   DATA[75,2] := 2.0;
   DATA[75,3] := 2.0;
   DATA[75,4] := 262.0161;
   DATA[75,5] := 8.391951;
   DATA[75,6] := 328.4286;
   DATA[75,7] := 2.440137;
   DATA[75,8] := 2.0;
   DATA[75,9] := 2.0;
   DATA[75,10] := 2.0;
   DATA[75,11] := 19.59472;
   DATA[75,12] := 2.21055;
   DATA[75,13] := 960.3307;
   DATA[75,14] := 1.0;
   DATA[75,15] := 2.0;
   DATA[75,16] := 1.0;
   DATA[75,17] := 1.0;
   DATA[75,18] := 1.0;
   DATA[75,19] := 2.0;
   DATA[75,20] := 148.808;
   DATA[75,21] := 156.242;
   DATA[75,22] := 1.720309;
   DATA[75,23] := 947.757;
   DATA[75,24] := 2.0;
   DATA[75,25] := 2.0;
   DATA[75,26] := 7.878621;
   DATA[75,27] := 145.0397;
   DATA[75,28] := 264.4194;
   DATA[75,29] := 12.03538;
   DATA[75,30] := 1.729428;
   DATA[75,31] := 1.291533;
   DATA[75,32] := 0.736421;
   DATA[75,33] := 0.3065689;
   DATA[75,34] := 2.0;
   DATA[75,35] := 251.2657;
   DATA[75,36] := 1.665972;
   DATA[75,37] := 189.9833;
   DATA[75,38] := 0.000128152;
   DATA[75,39] := 1.0;
   DATA[76,0] := 2.44179;
   DATA[76,1] := 524.6916;
   DATA[76,2] := 2.0;
   DATA[76,3] := 2.0;
   DATA[76,4] := 262.0161;
   DATA[76,5] := 8.391951;
   DATA[76,6] := 328.4286;
   DATA[76,7] := 2.440137;
   DATA[76,8] := 2.0;
   DATA[76,9] := 2.0;
   DATA[76,10] := 2.0;
   DATA[76,11] := 19.62354;
   DATA[76,12] := 2.21055;
   DATA[76,13] := 959.9702;
   DATA[76,14] := 1.0;
   DATA[76,15] := 2.0;
   DATA[76,16] := 1.0;
   DATA[76,17] := 1.0;
   DATA[76,18] := 1.0;
   DATA[76,19] := 2.0;
   DATA[76,20] := 148.808;
   DATA[76,21] := 156.242;
   DATA[76,22] := 1.719796;
   DATA[76,23] := 948.2184;
   DATA[76,24] := 2.0;
   DATA[76,25] := 2.0;
   DATA[76,26] := 7.878621;
   DATA[76,27] := 145.0397;
   DATA[76,28] := 264.4194;
   DATA[76,29] := 12.03538;
   DATA[76,30] := 1.726096;
   DATA[76,31] := 1.303446;
   DATA[76,32] := 0.736421;
   DATA[76,33] := 0.3065689;
   DATA[76,34] := 2.0;
   DATA[76,35] := 251.2657;
   DATA[76,36] := 1.665972;
   DATA[76,37] := 189.9833;
   DATA[76,38] := 0.000128152;
   DATA[76,39] := 1.0;
   DATA[77,0] := 2.431221;
   DATA[77,1] := 525.0842;
   DATA[77,2] := 2.0;
   DATA[77,3] := 2.0;
   DATA[77,4] := 262.0161;
   DATA[77,5] := 8.391951;
   DATA[77,6] := 328.4286;
   DATA[77,7] := 2.440137;
   DATA[77,8] := 2.0;
   DATA[77,9] := 2.0;
   DATA[77,10] := 2.0;
   DATA[77,11] := 19.64274;
   DATA[77,12] := 2.21055;
   DATA[77,13] := 960.0103;
   DATA[77,14] := 1.0;
   DATA[77,15] := 2.0;
   DATA[77,16] := 1.0;
   DATA[77,17] := 1.0;
   DATA[77,18] := 1.0;
   DATA[77,19] := 2.0;
   DATA[77,20] := 148.808;
   DATA[77,21] := 156.242;
   DATA[77,22] := 1.718515;
   DATA[77,23] := 948.6029;
   DATA[77,24] := 2.0;
   DATA[77,25] := 2.0;
   DATA[77,26] := 7.878621;
   DATA[77,27] := 145.0397;
   DATA[77,28] := 264.4194;
   DATA[77,29] := 12.03538;
   DATA[77,30] := 1.726096;
   DATA[77,31] := 1.311387;
   DATA[77,32] := 0.736421;
   DATA[77,33] := 0.3068891;
   DATA[77,34] := 2.0;
   DATA[77,35] := 250.9933;
   DATA[77,36] := 1.665972;
   DATA[77,37] := 189.8071;
   DATA[77,38] := 0.000128152;
   DATA[77,39] := 1.0;
   DATA[78,0] := 2.421932;
   DATA[78,1] := 525.2411;
   DATA[78,2] := 2.0;
   DATA[78,3] := 2.0;
   DATA[78,4] := 262.0161;
   DATA[78,5] := 8.391951;
   DATA[78,6] := 328.4286;
   DATA[78,7] := 2.440137;
   DATA[78,8] := 2.0;
   DATA[78,9] := 2.0;
   DATA[78,10] := 2.0;
   DATA[78,11] := 19.64274;
   DATA[78,12] := 2.208756;
   DATA[78,13] := 960.1304;
   DATA[78,14] := 1.0;
   DATA[78,15] := 2.0;
   DATA[78,16] := 1.0;
   DATA[78,17] := 1.0;
   DATA[78,18] := 1.0;
   DATA[78,19] := 2.0;
   DATA[78,20] := 148.808;
   DATA[78,21] := 156.242;
   DATA[78,22] := 1.718515;
   DATA[78,23] := 948.5645;
   DATA[78,24] := 2.0;
   DATA[78,25] := 2.0;
   DATA[78,26] := 7.878621;
   DATA[78,27] := 145.0397;
   DATA[78,28] := 264.2912;
   DATA[78,29] := 12.03538;
   DATA[78,30] := 1.725968;
   DATA[78,31] := 1.306008;
   DATA[78,32] := 0.736421;
   DATA[78,33] := 0.3068891;
   DATA[78,34] := 2.0;
   DATA[78,35] := 250.9933;
   DATA[78,36] := 1.665972;
   DATA[78,37] := 189.6629;
   DATA[78,38] := 0.000128152;
   DATA[78,39] := 1.0;
   DATA[79,0] := 2.420011;
   DATA[79,1] := 525.5159;
   DATA[79,2] := 2.0;
   DATA[79,3] := 2.0;
   DATA[79,4] := 262.0161;
   DATA[79,5] := 8.391951;
   DATA[79,6] := 328.4286;
   DATA[79,7] := 2.440137;
   DATA[79,8] := 2.0;
   DATA[79,9] := 2.0;
   DATA[79,10] := 2.0;
   DATA[79,11] := 19.64274;
   DATA[79,12] := 2.208756;
   DATA[79,13] := 959.9702;
   DATA[79,14] := 1.0;
   DATA[79,15] := 2.0;
   DATA[79,16] := 1.0;
   DATA[79,17] := 1.0;
   DATA[79,18] := 1.0;
   DATA[79,19] := 2.0;
   DATA[79,20] := 148.808;
   DATA[79,21] := 156.242;
   DATA[79,22] := 1.720309;
   DATA[79,23] := 948.7952;
   DATA[79,24] := 2.0;
   DATA[79,25] := 2.0;
   DATA[79,26] := 7.878621;
   DATA[79,27] := 145.1679;
   DATA[79,28] := 264.2912;
   DATA[79,29] := 12.03538;
   DATA[79,30] := 1.724814;
   DATA[79,31] := 1.306904;
   DATA[79,32] := 0.7353967;
   DATA[79,33] := 0.3068891;
   DATA[79,34] := 2.0;
   DATA[79,35] := 250.9933;
   DATA[79,36] := 1.665972;
   DATA[79,37] := 189.6629;
   DATA[79,38] := 0.000128152;
   DATA[79,39] := 1.0;
   DATA[80,0] := 2.447875;
   DATA[80,1] := 525.3196;
   DATA[80,2] := 2.0;
   DATA[80,3] := 2.0;
   DATA[80,4] := 262.0161;
   DATA[80,5] := 8.394835;
   DATA[80,6] := 328.4286;
   DATA[80,7] := 2.440137;
   DATA[80,8] := 2.0;
   DATA[80,9] := 2.0;
   DATA[80,10] := 2.0;
   DATA[80,11] := 19.65555;
   DATA[80,12] := 2.208756;
   DATA[80,13] := 960.3708;
   DATA[80,14] := 1.0;
   DATA[80,15] := 2.0;
   DATA[80,16] := 1.0;
   DATA[80,17] := 1.0;
   DATA[80,18] := 1.0;
   DATA[80,19] := 2.0;
   DATA[80,20] := 148.808;
   DATA[80,21] := 156.242;
   DATA[80,22] := 1.720309;
   DATA[80,23] := 948.9105;
   DATA[80,24] := 2.0;
   DATA[80,25] := 2.0;
   DATA[80,26] := 7.878621;
   DATA[80,27] := 145.2448;
   DATA[80,28] := 264.2912;
   DATA[80,29] := 12.03538;
   DATA[80,30] := 1.724814;
   DATA[80,31] := 1.297938;
   DATA[80,32] := 0.7353967;
   DATA[80,33] := 0.3068891;
   DATA[80,34] := 2.0;
   DATA[80,35] := 250.9933;
   DATA[80,36] := 1.665972;
   DATA[80,37] := 189.6629;
   DATA[80,38] := 0.000128152;
   DATA[80,39] := 1.0;
   DATA[81,0] := 2.500721;
   DATA[81,1] := 526.0262;
   DATA[81,2] := 2.0;
   DATA[81,3] := 2.0;
   DATA[81,4] := 262.0161;
   DATA[81,5] := 8.394835;
   DATA[81,6] := 328.4286;
   DATA[81,7] := 2.440137;
   DATA[81,8] := 2.0;
   DATA[81,9] := 2.0;
   DATA[81,10] := 2.0;
   DATA[81,11] := 19.65555;
   DATA[81,12] := 2.208756;
   DATA[81,13] := 960.2506;
   DATA[81,14] := 1.0;
   DATA[81,15] := 2.0;
   DATA[81,16] := 1.0;
   DATA[81,17] := 1.0;
   DATA[81,18] := 1.0;
   DATA[81,19] := 2.0;
   DATA[81,20] := 148.808;
   DATA[81,21] := 156.242;
   DATA[81,22] := 1.720309;
   DATA[81,23] := 949.1028;
   DATA[81,24] := 2.0;
   DATA[81,25] := 2.0;
   DATA[81,26] := 7.878621;
   DATA[81,27] := 145.2448;
   DATA[81,28] := 264.2592;
   DATA[81,29] := 12.03538;
   DATA[81,30] := 1.724814;
   DATA[81,31] := 1.292174;
   DATA[81,32] := 0.7353967;
   DATA[81,33] := 0.3066329;
   DATA[81,34] := 2.0;
   DATA[81,35] := 250.9933;
   DATA[81,36] := 1.569859;
   DATA[81,37] := 189.6629;
   DATA[81,38] := 0.000128152;
   DATA[81,39] := 1.0;
   DATA[82,0] := 2.543958;
   DATA[82,1] := 526.4973;
   DATA[82,2] := 2.0;
   DATA[82,3] := 2.0;
   DATA[82,4] := 262.0161;
   DATA[82,5] := 8.394835;
   DATA[82,6] := 328.4286;
   DATA[82,7] := 2.440137;
   DATA[82,8] := 2.0;
   DATA[82,9] := 2.0;
   DATA[82,10] := 2.0;
   DATA[82,11] := 19.65555;
   DATA[82,12] := 2.208756;
   DATA[82,13] := 960.0904;
   DATA[82,14] := 1.0;
   DATA[82,15] := 2.0;
   DATA[82,16] := 1.0;
   DATA[82,17] := 1.0;
   DATA[82,18] := 1.0;
   DATA[82,19] := 2.0;
   DATA[82,20] := 148.808;
   DATA[82,21] := 156.242;
   DATA[82,22] := 1.718643;
   DATA[82,23] := 949.1797;
   DATA[82,24] := 2.0;
   DATA[82,25] := 2.0;
   DATA[82,26] := 7.878621;
   DATA[82,27] := 145.2448;
   DATA[82,28] := 264.2592;
   DATA[82,29] := 12.03538;
   DATA[82,30] := 1.724814;
   DATA[82,31] := 1.288971;
   DATA[82,32] := 0.7353967;
   DATA[82,33] := 0.3065048;
   DATA[82,34] := 2.0;
   DATA[82,35] := 250.9933;
   DATA[82,36] := 1.569859;
   DATA[82,37] := 189.6629;
   DATA[82,38] := 0.000128152;
   DATA[82,39] := 1.0;
   DATA[83,0] := 2.570861;
   DATA[83,1] := 526.8898;
   DATA[83,2] := 2.0;
   DATA[83,3] := 2.0;
   DATA[83,4] := 262.0161;
   DATA[83,5] := 8.394835;
   DATA[83,6] := 328.4286;
   DATA[83,7] := 2.441034;
   DATA[83,8] := 2.0;
   DATA[83,9] := 2.0;
   DATA[83,10] := 2.0;
   DATA[83,11] := 19.65555;
   DATA[83,12] := 2.208756;
   DATA[83,13] := 959.8901;
   DATA[83,14] := 1.0;
   DATA[83,15] := 2.0;
   DATA[83,16] := 1.0;
   DATA[83,17] := 1.0;
   DATA[83,18] := 1.0;
   DATA[83,19] := 2.0;
   DATA[83,20] := 148.808;
   DATA[83,21] := 156.242;
   DATA[83,22] := 1.718643;
   DATA[83,23] := 949.2181;
   DATA[83,24] := 2.0;
   DATA[83,25] := 2.0;
   DATA[83,26] := 7.878621;
   DATA[83,27] := 145.2448;
   DATA[83,28] := 264.2592;
   DATA[83,29] := 12.03538;
   DATA[83,30] := 1.724814;
   DATA[83,31] := 1.282311;
   DATA[83,32] := 0.7353967;
   DATA[83,33] := 0.3065048;
   DATA[83,34] := 2.0;
   DATA[83,35] := 250.9933;
   DATA[83,36] := 1.569859;
   DATA[83,37] := 189.6629;
   DATA[83,38] := 0.000128152;
   DATA[83,39] := 1.0;
   DATA[84,0] := 2.614739;
   DATA[84,1] := 527.2038;
   DATA[84,2] := 2.0;
   DATA[84,3] := 2.0;
   DATA[84,4] := 262.0161;
   DATA[84,5] := 8.394835;
   DATA[84,6] := 328.4286;
   DATA[84,7] := 2.441034;
   DATA[84,8] := 2.0;
   DATA[84,9] := 2.0;
   DATA[84,10] := 2.0;
   DATA[84,11] := 19.65555;
   DATA[84,12] := 2.208756;
   DATA[84,13] := 959.8901;
   DATA[84,14] := 1.0;
   DATA[84,15] := 2.0;
   DATA[84,16] := 1.0;
   DATA[84,17] := 1.0;
   DATA[84,18] := 1.0;
   DATA[84,19] := 2.0;
   DATA[84,20] := 148.808;
   DATA[84,21] := 156.242;
   DATA[84,22] := 1.718643;
   DATA[84,23] := 949.8718;
   DATA[84,24] := 2.0;
   DATA[84,25] := 2.0;
   DATA[84,26] := 7.878621;
   DATA[84,27] := 145.1423;
   DATA[84,28] := 264.2592;
   DATA[84,29] := 12.03538;
   DATA[84,30] := 1.724814;
   DATA[84,31] := 1.27898;
   DATA[84,32] := 0.7353967;
   DATA[84,33] := 0.3065048;
   DATA[84,34] := 2.0;
   DATA[84,35] := 250.9933;
   DATA[84,36] := 1.569859;
   DATA[84,37] := 189.6629;
   DATA[84,38] := 0.000128152;
   DATA[84,39] := 1.0;
   DATA[85,0] := 2.645806;
   DATA[85,1] := 527.3608;
   DATA[85,2] := 2.0;
   DATA[85,3] := 2.0;
   DATA[85,4] := 262.2084;
   DATA[85,5] := 8.394835;
   DATA[85,6] := 328.4286;
   DATA[85,7] := 2.441034;
   DATA[85,8] := 2.0;
   DATA[85,9] := 2.0;
   DATA[85,10] := 2.0;
   DATA[85,11] := 19.65555;
   DATA[85,12] := 2.208756;
   DATA[85,13] := 960.0103;
   DATA[85,14] := 1.0;
   DATA[85,15] := 2.0;
   DATA[85,16] := 1.0;
   DATA[85,17] := 1.0;
   DATA[85,18] := 1.0;
   DATA[85,19] := 2.0;
   DATA[85,20] := 148.808;
   DATA[85,21] := 156.0882;
   DATA[85,22] := 1.720693;
   DATA[85,23] := 950.0641;
   DATA[85,24] := 2.0;
   DATA[85,25] := 2.0;
   DATA[85,26] := 7.878621;
   DATA[85,27] := 144.9885;
   DATA[85,28] := 264.2592;
   DATA[85,29] := 12.03538;
   DATA[85,30] := 1.724814;
   DATA[85,31] := 1.27232;
   DATA[85,32] := 0.7353967;
   DATA[85,33] := 0.3065048;
   DATA[85,34] := 2.0;
   DATA[85,35] := 250.9933;
   DATA[85,36] := 1.569859;
   DATA[85,37] := 189.7751;
   DATA[85,38] := 0.000128152;
   DATA[85,39] := 1.0;
   DATA[86,0] := 2.665023;
   DATA[86,1] := 527.4786;
   DATA[86,2] := 2.0;
   DATA[86,3] := 2.0;
   DATA[86,4] := 262.2084;
   DATA[86,5] := 8.394835;
   DATA[86,6] := 328.4286;
   DATA[86,7] := 2.441034;
   DATA[86,8] := 2.0;
   DATA[86,9] := 2.0;
   DATA[86,10] := 2.0;
   DATA[86,11] := 19.65555;
   DATA[86,12] := 2.208756;
   DATA[86,13] := 959.8901;
   DATA[86,14] := 1.0;
   DATA[86,15] := 2.0;
   DATA[86,16] := 1.0;
   DATA[86,17] := 1.0;
   DATA[86,18] := 1.0;
   DATA[86,19] := 2.0;
   DATA[86,20] := 148.808;
   DATA[86,21] := 156.0882;
   DATA[86,22] := 1.720693;
   DATA[86,23] := 950.1794;
   DATA[86,24] := 2.0;
   DATA[86,25] := 2.0;
   DATA[86,26] := 7.878621;
   DATA[86,27] := 144.9885;
   DATA[86,28] := 264.2592;
   DATA[86,29] := 12.03538;
   DATA[86,30] := 1.724814;
   DATA[86,31] := 1.270398;
   DATA[86,32] := 0.7353967;
   DATA[86,33] := 0.3065048;
   DATA[86,34] := 2.0;
   DATA[86,35] := 250.9933;
   DATA[86,36] := 1.569859;
   DATA[86,37] := 189.7751;
   DATA[86,38] := 0.000128152;
   DATA[86,39] := 1.0;
   DATA[87,0] := 2.666944;
   DATA[87,1] := 527.7534;
   DATA[87,2] := 2.0;
   DATA[87,3] := 2.0;
   DATA[87,4] := 262.2084;
   DATA[87,5] := 8.393553;
   DATA[87,6] := 328.4286;
   DATA[87,7] := 2.441547;
   DATA[87,8] := 2.0;
   DATA[87,9] := 2.0;
   DATA[87,10] := 2.0;
   DATA[87,11] := 19.65555;
   DATA[87,12] := 2.208756;
   DATA[87,13] := 959.5296;
   DATA[87,14] := 1.0;
   DATA[87,15] := 2.0;
   DATA[87,16] := 1.0;
   DATA[87,17] := 1.0;
   DATA[87,18] := 1.0;
   DATA[87,19] := 2.0;
   DATA[87,20] := 148.808;
   DATA[87,21] := 156.0882;
   DATA[87,22] := 1.720693;
   DATA[87,23] := 950.0641;
   DATA[87,24] := 2.0;
   DATA[87,25] := 2.0;
   DATA[87,26] := 7.878621;
   DATA[87,27] := 144.9885;
   DATA[87,28] := 264.2592;
   DATA[87,29] := 12.30454;
   DATA[87,30] := 1.724814;
   DATA[87,31] := 1.270398;
   DATA[87,32] := 0.7353967;
   DATA[87,33] := 0.3065048;
   DATA[87,34] := 2.0;
   DATA[87,35] := 250.9933;
   DATA[87,36] := 1.569859;
   DATA[87,37] := 189.7751;
   DATA[87,38] := 0.000128152;
   DATA[87,39] := 1.0;
   DATA[88,0] := 2.6394;
   DATA[88,1] := 528.2244;
   DATA[88,2] := 2.0;
   DATA[88,3] := 2.0;
   DATA[88,4] := 262.2084;
   DATA[88,5] := 8.391951;
   DATA[88,6] := 328.4286;
   DATA[88,7] := 2.443597;
   DATA[88,8] := 2.0;
   DATA[88,9] := 2.0;
   DATA[88,10] := 2.0;
   DATA[88,11] := 19.65555;
   DATA[88,12] := 2.209653;
   DATA[88,13] := 959.4896;
   DATA[88,14] := 1.0;
   DATA[88,15] := 2.0;
   DATA[88,16] := 1.0;
   DATA[88,17] := 1.0;
   DATA[88,18] := 1.0;
   DATA[88,19] := 2.0;
   DATA[88,20] := 148.808;
   DATA[88,21] := 156.0882;
   DATA[88,22] := 1.720693;
   DATA[88,23] := 950.2563;
   DATA[88,24] := 2.0;
   DATA[88,25] := 2.0;
   DATA[88,26] := 7.878621;
   DATA[88,27] := 144.9885;
   DATA[88,28] := 264.2592;
   DATA[88,29] := 12.30454;
   DATA[88,30] := 1.727378;
   DATA[88,31] := 1.284232;
   DATA[88,32] := 0.7353967;
   DATA[88,33] := 0.3065048;
   DATA[88,34] := 2.0;
   DATA[88,35] := 250.9933;
   DATA[88,36] := 1.569859;
   DATA[88,37] := 189.7751;
   DATA[88,38] := 0.000128152;
   DATA[88,39] := 1.0;
   DATA[89,0] := 2.620824;
   DATA[89,1] := 527.8711;
   DATA[89,2] := 2.0;
   DATA[89,3] := 2.0;
   DATA[89,4] := 261.9841;
   DATA[89,5] := 8.391951;
   DATA[89,6] := 328.4286;
   DATA[89,7] := 2.444751;
   DATA[89,8] := 2.0;
   DATA[89,9] := 2.0;
   DATA[89,10] := 2.0;
   DATA[89,11] := 19.60433;
   DATA[89,12] := 2.209653;
   DATA[89,13] := 959.5697;
   DATA[89,14] := 1.0;
   DATA[89,15] := 2.0;
   DATA[89,16] := 1.0;
   DATA[89,17] := 1.0;
   DATA[89,18] := 1.0;
   DATA[89,19] := 2.0;
   DATA[89,20] := 148.808;
   DATA[89,21] := 156.0882;
   DATA[89,22] := 1.719924;
   DATA[89,23] := 950.5255;
   DATA[89,24] := 2.0;
   DATA[89,25] := 2.0;
   DATA[89,26] := 7.878621;
   DATA[89,27] := 144.9885;
   DATA[89,28] := 264.2592;
   DATA[89,29] := 12.30454;
   DATA[89,30] := 1.727378;
   DATA[89,31] := 1.290765;
   DATA[89,32] := 0.7353967;
   DATA[89,33] := 0.3065048;
   DATA[89,34] := 2.0;
   DATA[89,35] := 250.9933;
   DATA[89,36] := 1.569859;
   DATA[89,37] := 189.7751;
   DATA[89,38] := 0.000128152;
   DATA[89,39] := 1.0;
   DATA[90,0] := 2.61634;
   DATA[90,1] := 528.0281;
   DATA[90,2] := 2.0;
   DATA[90,3] := 2.0;
   DATA[90,4] := 261.9841;
   DATA[90,5] := 8.391951;
   DATA[90,6] := 328.4286;
   DATA[90,7] := 2.444751;
   DATA[90,8] := 2.0;
   DATA[90,9] := 2.0;
   DATA[90,10] := 2.0;
   DATA[90,11] := 19.60433;
   DATA[90,12] := 2.209653;
   DATA[90,13] := 959.5697;
   DATA[90,14] := 1.0;
   DATA[90,15] := 2.0;
   DATA[90,16] := 1.0;
   DATA[90,17] := 1.0;
   DATA[90,18] := 1.0;
   DATA[90,19] := 2.0;
   DATA[90,20] := 148.808;
   DATA[90,21] := 156.0882;
   DATA[90,22] := 1.719284;
   DATA[90,23] := 950.6409;
   DATA[90,24] := 2.0;
   DATA[90,25] := 2.0;
   DATA[90,26] := 7.878621;
   DATA[90,27] := 145.1166;
   DATA[90,28] := 264.2592;
   DATA[90,29] := 12.30454;
   DATA[90,30] := 1.727378;
   DATA[90,31] := 1.285385;
   DATA[90,32] := 0.7353967;
   DATA[90,33] := 0.3065048;
   DATA[90,34] := 2.0;
   DATA[90,35] := 250.9933;
   DATA[90,36] := 1.681991;
   DATA[90,37] := 189.7751;
   DATA[90,38] := 0.000128152;
   DATA[90,39] := 1.0;
   DATA[91,0] := 2.61602;
   DATA[91,1] := 527.7534;
   DATA[91,2] := 2.0;
   DATA[91,3] := 2.0;
   DATA[91,4] := 261.9841;
   DATA[91,5] := 8.391951;
   DATA[91,6] := 328.4286;
   DATA[91,7] := 2.444751;
   DATA[91,8] := 2.0;
   DATA[91,9] := 2.0;
   DATA[91,10] := 2.0;
   DATA[91,11] := 19.60433;
   DATA[91,12] := 2.212215;
   DATA[91,13] := 959.4095;
   DATA[91,14] := 1.0;
   DATA[91,15] := 2.0;
   DATA[91,16] := 1.0;
   DATA[91,17] := 1.0;
   DATA[91,18] := 1.0;
   DATA[91,19] := 2.0;
   DATA[91,20] := 148.808;
   DATA[91,21] := 156.0882;
   DATA[91,22] := 1.719284;
   DATA[91,23] := 950.8331;
   DATA[91,24] := 2.0;
   DATA[91,25] := 2.0;
   DATA[91,26] := 7.878621;
   DATA[91,27] := 145.1679;
   DATA[91,28] := 264.2592;
   DATA[91,29] := 12.30454;
   DATA[91,30] := 1.727378;
   DATA[91,31] := 1.288843;
   DATA[91,32] := 0.7353967;
   DATA[91,33] := 0.3065048;
   DATA[91,34] := 2.0;
   DATA[91,35] := 250.9933;
   DATA[91,36] := 1.681991;
   DATA[91,37] := 189.7751;
   DATA[91,38] := 0.000128152;
   DATA[91,39] := 1.0;
   DATA[92,0] := 2.609294;
   DATA[92,1] := 527.4393;
   DATA[92,2] := 2.0;
   DATA[92,3] := 2.0;
   DATA[92,4] := 261.9841;
   DATA[92,5] := 8.391951;
   DATA[92,6] := 328.4286;
   DATA[92,7] := 2.443085;
   DATA[92,8] := 2.0;
   DATA[92,9] := 2.0;
   DATA[92,10] := 2.0;
   DATA[92,11] := 19.64274;
   DATA[92,12] := 2.212215;
   DATA[92,13] := 959.77;
   DATA[92,14] := 1.0;
   DATA[92,15] := 2.0;
   DATA[92,16] := 1.0;
   DATA[92,17] := 1.0;
   DATA[92,18] := 1.0;
   DATA[92,19] := 2.0;
   DATA[92,20] := 148.808;
   DATA[92,21] := 156.0882;
   DATA[92,22] := 1.718387;
   DATA[92,23] := 950.8716;
   DATA[92,24] := 2.0;
   DATA[92,25] := 2.0;
   DATA[92,26] := 7.878621;
   DATA[92,27] := 145.1679;
   DATA[92,28] := 264.2592;
   DATA[92,29] := 12.30454;
   DATA[92,30] := 1.727378;
   DATA[92,31] := 1.278468;
   DATA[92,32] := 0.7353967;
   DATA[92,33] := 0.3065048;
   DATA[92,34] := 2.0;
   DATA[92,35] := 250.9933;
   DATA[92,36] := 1.681991;
   DATA[92,37] := 189.7751;
   DATA[92,38] := 0.000128152;
   DATA[92,39] := 1.0;
   DATA[93,0] := 2.584313;
   DATA[93,1] := 527.2823;
   DATA[93,2] := 2.0;
   DATA[93,3] := 2.0;
   DATA[93,4] := 261.9841;
   DATA[93,5] := 8.391951;
   DATA[93,6] := 328.4286;
   DATA[93,7] := 2.442316;
   DATA[93,8] := 2.0;
   DATA[93,9] := 2.0;
   DATA[93,10] := 2.0;
   DATA[93,11] := 19.65875;
   DATA[93,12] := 2.212343;
   DATA[93,13] := 960.0904;
   DATA[93,14] := 1.0;
   DATA[93,15] := 2.0;
   DATA[93,16] := 1.0;
   DATA[93,17] := 1.0;
   DATA[93,18] := 1.0;
   DATA[93,19] := 2.0;
   DATA[93,20] := 148.808;
   DATA[93,21] := 156.0882;
   DATA[93,22] := 1.716849;
   DATA[93,23] := 951.0638;
   DATA[93,24] := 2.0;
   DATA[93,25] := 2.0;
   DATA[93,26] := 7.877019;
   DATA[93,27] := 145.1679;
   DATA[93,28] := 264.2592;
   DATA[93,29] := 12.30454;
   DATA[93,30] := 1.727378;
   DATA[93,31] := 1.263097;
   DATA[93,32] := 0.7353967;
   DATA[93,33] := 0.3065048;
   DATA[93,34] := 2.0;
   DATA[93,35] := 251.1055;
   DATA[93,36] := 1.649953;
   DATA[93,37] := 189.7751;
   DATA[93,38] := 0.000128152;
   DATA[93,39] := 1.0;
   DATA[94,0] := 2.572463;
   DATA[94,1] := 527.2823;
   DATA[94,2] := 2.0;
   DATA[94,3] := 2.0;
   DATA[94,4] := 261.9841;
   DATA[94,5] := 8.391951;
   DATA[94,6] := 328.4286;
   DATA[94,7] := 2.442188;
   DATA[94,8] := 2.0;
   DATA[94,9] := 2.0;
   DATA[94,10] := 2.0;
   DATA[94,11] := 19.65875;
   DATA[94,12] := 2.212343;
   DATA[94,13] := 960.0103;
   DATA[94,14] := 1.0;
   DATA[94,15] := 2.0;
   DATA[94,16] := 1.0;
   DATA[94,17] := 1.0;
   DATA[94,18] := 1.0;
   DATA[94,19] := 2.0;
   DATA[94,20] := 148.808;
   DATA[94,21] := 156.0882;
   DATA[94,22] := 1.714029;
   DATA[94,23] := 950.8331;
   DATA[94,24] := 2.0;
   DATA[94,25] := 2.0;
   DATA[94,26] := 7.877019;
   DATA[94,27] := 145.1423;
   DATA[94,28] := 264.2592;
   DATA[94,29] := 12.30454;
   DATA[94,30] := 1.727378;
   DATA[94,31] := 1.257589;
   DATA[94,32] := 0.7353967;
   DATA[94,33] := 0.3065048;
   DATA[94,34] := 2.0;
   DATA[94,35] := 251.1055;
   DATA[94,36] := 1.649953;
   DATA[94,37] := 189.7751;
   DATA[94,38] := 0.000128152;
   DATA[94,39] := 1.0;
   DATA[95,0] := 2.554847;
   DATA[95,1] := 527.3608;
   DATA[95,2] := 2.0;
   DATA[95,3] := 2.0;
   DATA[95,4] := 261.9841;
   DATA[95,5] := 8.391951;
   DATA[95,6] := 328.4286;
   DATA[95,7] := 2.442188;
   DATA[95,8] := 2.0;
   DATA[95,9] := 2.0;
   DATA[95,10] := 2.0;
   DATA[95,11] := 19.65875;
   DATA[95,12] := 2.212343;
   DATA[95,13] := 959.9302;
   DATA[95,14] := 1.0;
   DATA[95,15] := 2.0;
   DATA[95,16] := 1.0;
   DATA[95,17] := 1.0;
   DATA[95,18] := 1.0;
   DATA[95,19] := 2.0;
   DATA[95,20] := 148.808;
   DATA[95,21] := 156.0882;
   DATA[95,22] := 1.713261;
   DATA[95,23] := 950.91;
   DATA[95,24] := 2.0;
   DATA[95,25] := 2.0;
   DATA[95,26] := 7.877019;
   DATA[95,27] := 145.1423;
   DATA[95,28] := 264.2592;
   DATA[95,29] := 12.30454;
   DATA[95,30] := 1.727378;
   DATA[95,31] := 1.245549;
   DATA[95,32] := 0.7353967;
   DATA[95,33] := 0.3065048;
   DATA[95,34] := 2.0;
   DATA[95,35] := 251.1055;
   DATA[95,36] := 1.649953;
   DATA[95,37] := 189.7751;
   DATA[95,38] := 0.000128152;
   DATA[95,39] := 1.0;
   DATA[96,0] := 2.542036;
   DATA[96,1] := 526.8113;
   DATA[96,2] := 2.0;
   DATA[96,3] := 2.0;
   DATA[96,4] := 261.9841;
   DATA[96,5] := 8.39163;
   DATA[96,6] := 328.4286;
   DATA[96,7] := 2.442188;
   DATA[96,8] := 2.0;
   DATA[96,9] := 2.0;
   DATA[96,10] := 2.0;
   DATA[96,11] := 19.64594;
   DATA[96,12] := 2.212343;
   DATA[96,13] := 960.2506;
   DATA[96,14] := 1.0;
   DATA[96,15] := 2.0;
   DATA[96,16] := 1.0;
   DATA[96,17] := 1.0;
   DATA[96,18] := 1.0;
   DATA[96,19] := 2.0;
   DATA[96,20] := 148.808;
   DATA[96,21] := 156.0882;
   DATA[96,22] := 1.712876;
   DATA[96,23] := 951.2561;
   DATA[96,24] := 2.0;
   DATA[96,25] := 2.0;
   DATA[96,26] := 7.877019;
   DATA[96,27] := 144.9628;
   DATA[96,28] := 264.2592;
   DATA[96,29] := 12.11228;
   DATA[96,30] := 1.726865;
   DATA[96,31] := 1.256693;
   DATA[96,32] := 0.7353967;
   DATA[96,33] := 0.3065048;
   DATA[96,34] := 2.0;
   DATA[96,35] := 251.1055;
   DATA[96,36] := 1.649953;
   DATA[96,37] := 189.7751;
   DATA[96,38] := 0.000128152;
   DATA[96,39] := 1.0;
   DATA[97,0] := 2.520257;
   DATA[97,1] := 526.5757;
   DATA[97,2] := 2.0;
   DATA[97,3] := 2.0;
   DATA[97,4] := 261.9841;
   DATA[97,5] := 8.39163;
   DATA[97,6] := 328.4286;
   DATA[97,7] := 2.442188;
   DATA[97,8] := 2.0;
   DATA[97,9] := 2.0;
   DATA[97,10] := 2.0;
   DATA[97,11] := 19.62354;
   DATA[97,12] := 2.212343;
   DATA[97,13] := 960.531;
   DATA[97,14] := 1.0;
   DATA[97,15] := 2.0;
   DATA[97,16] := 1.0;
   DATA[97,17] := 1.0;
   DATA[97,18] := 1.0;
   DATA[97,19] := 2.0;
   DATA[97,20] := 148.808;
   DATA[97,21] := 156.0882;
   DATA[97,22] := 1.713261;
   DATA[97,23] := 951.2561;
   DATA[97,24] := 2.0;
   DATA[97,25] := 2.0;
   DATA[97,26] := 7.877019;
   DATA[97,27] := 144.8603;
   DATA[97,28] := 264.2592;
   DATA[97,29] := 12.07383;
   DATA[97,30] := 1.726865;
   DATA[97,31] := 1.265787;
   DATA[97,32] := 0.7353967;
   DATA[97,33] := 0.3074656;
   DATA[97,34] := 2.0;
   DATA[97,35] := 250.9773;
   DATA[97,36] := 1.649953;
   DATA[97,37] := 189.6789;
   DATA[97,38] := 0.000128152;
   DATA[97,39] := 1.0;
   DATA[98,0] := 2.508407;
   DATA[98,1] := 525.8692;
   DATA[98,2] := 2.0;
   DATA[98,3] := 2.0;
   DATA[98,4] := 261.9841;
   DATA[98,5] := 8.39163;
   DATA[98,6] := 328.4286;
   DATA[98,7] := 2.443469;
   DATA[98,8] := 2.0;
   DATA[98,9] := 2.0;
   DATA[98,10] := 2.0;
   DATA[98,11] := 19.62354;
   DATA[98,12] := 2.21055;
   DATA[98,13] := 960.3307;
   DATA[98,14] := 1.0;
   DATA[98,15] := 2.0;
   DATA[98,16] := 1.0;
   DATA[98,17] := 1.0;
   DATA[98,18] := 1.0;
   DATA[98,19] := 2.0;
   DATA[98,20] := 148.808;
   DATA[98,21] := 156.0882;
   DATA[98,22] := 1.715311;
   DATA[98,23] := 951.4099;
   DATA[98,24] := 2.0;
   DATA[98,25] := 2.0;
   DATA[98,26] := 7.877019;
   DATA[98,27] := 144.8603;
   DATA[98,28] := 264.2592;
   DATA[98,29] := 12.07383;
   DATA[98,30] := 1.725583;
   DATA[98,31] := 1.277956;
   DATA[98,32] := 0.7353967;
   DATA[98,33] := 0.3081062;
   DATA[98,34] := 2.0;
   DATA[98,35] := 250.8171;
   DATA[98,36] := 1.649953;
   DATA[98,37] := 189.5027;
   DATA[98,38] := 0.000128152;
   DATA[98,39] := 1.0;
   DATA[99,0] := 2.491112;
   DATA[99,1] := 525.3982;
   DATA[99,2] := 2.0;
   DATA[99,3] := 2.0;
   DATA[99,4] := 261.9841;
   DATA[99,5] := 8.39163;
   DATA[99,6] := 328.4286;
   DATA[99,7] := 2.444751;
   DATA[99,8] := 2.0;
   DATA[99,9] := 2.0;
   DATA[99,10] := 2.0;
   DATA[99,11] := 19.66195;
   DATA[99,12] := 2.209525;
   DATA[99,13] := 960.2106;
   DATA[99,14] := 1.0;
   DATA[99,15] := 2.0;
   DATA[99,16] := 1.0;
   DATA[99,17] := 1.0;
   DATA[99,18] := 1.0;
   DATA[99,19] := 2.0;
   DATA[99,20] := 148.808;
   DATA[99,21] := 156.1907;
   DATA[99,22] := 1.715311;
   DATA[99,23] := 951.2561;
   DATA[99,24] := 2.0;
   DATA[99,25] := 2.0;
   DATA[99,26] := 7.877019;
   DATA[99,27] := 144.8603;
   DATA[99,28] := 264.2592;
   DATA[99,29] := 12.07383;
   DATA[99,30] := 1.725455;
   DATA[99,31] := 1.289484;
   DATA[99,32] := 0.7378293;
   DATA[99,33] := 0.3081062;
   DATA[99,34] := 2.0;
   DATA[99,35] := 250.8171;
   DATA[99,36] := 1.649953;
   DATA[99,37] := 189.5027;
   DATA[99,38] := 0.000128152;
   DATA[99,39] := 1.0;
   DATA[100,0] := 2.476059;
   DATA[100,1] := 525.0842;
   DATA[100,2] := 2.0;
   DATA[100,3] := 2.0;
   DATA[100,4] := 261.9841;
   DATA[100,5] := 8.39163;
   DATA[100,6] := 328.4286;
   DATA[100,7] := 2.444751;
   DATA[100,8] := 2.0;
   DATA[100,9] := 2.0;
   DATA[100,10] := 2.0;
   DATA[100,11] := 19.66195;
   DATA[100,12] := 2.209525;
   DATA[100,13] := 960.3708;
   DATA[100,14] := 1.0;
   DATA[100,15] := 2.0;
   DATA[100,16] := 1.0;
   DATA[100,17] := 1.0;
   DATA[100,18] := 1.0;
   DATA[100,19] := 2.0;
   DATA[100,20] := 148.808;
   DATA[100,21] := 156.1907;
   DATA[100,22] := 1.715311;
   DATA[100,23] := 951.6791;
   DATA[100,24] := 2.0;
   DATA[100,25] := 2.0;
   DATA[100,26] := 7.877019;
   DATA[100,27] := 145.0397;
   DATA[100,28] := 264.2592;
   DATA[100,29] := 12.07383;
   DATA[100,30] := 1.723404;
   DATA[100,31] := 1.286666;
   DATA[100,32] := 0.7378293;
   DATA[100,33] := 0.3084265;
   DATA[100,34] := 2.0;
   DATA[100,35] := 250.8011;
   DATA[100,36] := 1.649953;
   DATA[100,37] := 189.5027;
   DATA[100,38] := 0.000128152;
   DATA[100,39] := 1.0;
   DATA[101,0] := 2.460045;
   DATA[101,1] := 524.8879;
   DATA[101,2] := 2.0;
   DATA[101,3] := 2.0;
   DATA[101,4] := 261.9841;
   DATA[101,5] := 8.39163;
   DATA[101,6] := 328.4286;
   DATA[101,7] := 2.444751;
   DATA[101,8] := 2.0;
   DATA[101,9] := 2.0;
   DATA[101,10] := 2.0;
   DATA[101,11] := 19.55631;
   DATA[101,12] := 2.209525;
   DATA[101,13] := 960.2106;
   DATA[101,14] := 1.0;
   DATA[101,15] := 2.0;
   DATA[101,16] := 1.0;
   DATA[101,17] := 1.0;
   DATA[101,18] := 1.0;
   DATA[101,19] := 2.0;
   DATA[101,20] := 148.808;
   DATA[101,21] := 156.1907;
   DATA[101,22] := 1.717105;
   DATA[101,23] := 951.9867;
   DATA[101,24] := 2.0;
   DATA[101,25] := 2.0;
   DATA[101,26] := 7.877019;
   DATA[101,27] := 145.0397;
   DATA[101,28] := 264.2592;
   DATA[101,29] := 12.07383;
   DATA[101,30] := 1.723404;
   DATA[101,31] := 1.293455;
   DATA[101,32] := 0.7360369;
   DATA[101,33] := 0.3086186;
   DATA[101,34] := 2.0;
   DATA[101,35] := 250.8011;
   DATA[101,36] := 1.649953;
   DATA[101,37] := 189.5027;
   DATA[101,38] := 0.000128152;
   DATA[101,39] := 1.0;
   DATA[102,0] := 2.445953;
   DATA[102,1] := 524.4561;
   DATA[102,2] := 2.0;
   DATA[102,3] := 2.0;
   DATA[102,4] := 261.9841;
   DATA[102,5] := 8.39163;
   DATA[102,6] := 328.4286;
   DATA[102,7] := 2.444751;
   DATA[102,8] := 2.0;
   DATA[102,9] := 2.0;
   DATA[102,10] := 2.0;
   DATA[102,11] := 19.50509;
   DATA[102,12] := 2.209525;
   DATA[102,13] := 960.2506;
   DATA[102,14] := 1.0;
   DATA[102,15] := 2.0;
   DATA[102,16] := 1.0;
   DATA[102,17] := 1.0;
   DATA[102,18] := 1.0;
   DATA[102,19] := 2.0;
   DATA[102,20] := 148.808;
   DATA[102,21] := 156.1907;
   DATA[102,22] := 1.717361;
   DATA[102,23] := 952.179;
   DATA[102,24] := 2.0;
   DATA[102,25] := 2.0;
   DATA[102,26] := 7.877019;
   DATA[102,27] := 145.0397;
   DATA[102,28] := 264.2592;
   DATA[102,29] := 12.07383;
   DATA[102,30] := 1.724942;
   DATA[102,31] := 1.289484;
   DATA[102,32] := 0.7353967;
   DATA[102,33] := 0.3086186;
   DATA[102,34] := 2.0;
   DATA[102,35] := 250.8011;
   DATA[102,36] := 1.649953;
   DATA[102,37] := 189.5027;
   DATA[102,38] := 0.000128152;
   DATA[102,39] := 1.0;
   DATA[103,0] := 2.42994;
   DATA[103,1] := 524.1028;
   DATA[103,2] := 2.0;
   DATA[103,3] := 2.0;
   DATA[103,4] := 261.9841;
   DATA[103,5] := 8.39163;
   DATA[103,6] := 328.4286;
   DATA[103,7] := 2.444751;
   DATA[103,8] := 2.0;
   DATA[103,9] := 2.0;
   DATA[103,10] := 2.0;
   DATA[103,11] := 19.50509;
   DATA[103,12] := 2.209525;
   DATA[103,13] := 960.4509;
   DATA[103,14] := 1.0;
   DATA[103,15] := 2.0;
   DATA[103,16] := 1.0;
   DATA[103,17] := 1.0;
   DATA[103,18] := 1.0;
   DATA[103,19] := 2.0;
   DATA[103,20] := 148.808;
   DATA[103,21] := 156.1907;
   DATA[103,22] := 1.717361;
   DATA[103,23] := 952.3712;
   DATA[103,24] := 2.0;
   DATA[103,25] := 2.0;
   DATA[103,26] := 7.877019;
   DATA[103,27] := 145.0397;
   DATA[103,28] := 264.2592;
   DATA[103,29] := 12.07383;
   DATA[103,30] := 1.725583;
   DATA[103,31] := 1.27232;
   DATA[103,32] := 0.7353967;
   DATA[103,33] := 0.3086186;
   DATA[103,34] := 2.0;
   DATA[103,35] := 251.0414;
   DATA[103,36] := 1.649953;
   DATA[103,37] := 189.6469;
   DATA[103,38] := 0.000128152;
   DATA[103,39] := 1.0;
   DATA[104,0] := 2.428658;
   DATA[104,1] := 524.0636;
   DATA[104,2] := 2.0;
   DATA[104,3] := 2.0;
   DATA[104,4] := 261.9841;
   DATA[104,5] := 8.39163;
   DATA[104,6] := 328.4286;
   DATA[104,7] := 2.444751;
   DATA[104,8] := 2.0;
   DATA[104,9] := 2.0;
   DATA[104,10] := 2.0;
   DATA[104,11] := 19.59793;
   DATA[104,12] := 2.209525;
   DATA[104,13] := 960.4108;
   DATA[104,14] := 1.0;
   DATA[104,15] := 2.0;
   DATA[104,16] := 1.0;
   DATA[104,17] := 1.0;
   DATA[104,18] := 1.0;
   DATA[104,19] := 2.0;
   DATA[104,20] := 148.808;
   DATA[104,21] := 156.1907;
   DATA[104,22] := 1.717361;
   DATA[104,23] := 952.4097;
   DATA[104,24] := 2.0;
   DATA[104,25] := 2.0;
   DATA[104,26] := 7.877019;
   DATA[104,27] := 145.0397;
   DATA[104,28] := 264.2592;
   DATA[104,29] := 12.07383;
   DATA[104,30] := 1.725583;
   DATA[104,31] := 1.260664;
   DATA[104,32] := 0.7353967;
   DATA[104,33] := 0.3086186;
   DATA[104,34] := 2.0;
   DATA[104,35] := 251.0414;
   DATA[104,36] := 1.649953;
   DATA[104,37] := 189.8071;
   DATA[104,38] := 0.000128152;
   DATA[104,39] := 1.0;
   DATA[105,0] := 2.426737;
   DATA[105,1] := 523.8673;
   DATA[105,2] := 2.0;
   DATA[105,3] := 2.0;
   DATA[105,4] := 262.1764;
   DATA[105,5] := 8.39163;
   DATA[105,6] := 328.4286;
   DATA[105,7] := 2.444751;
   DATA[105,8] := 2.0;
   DATA[105,9] := 2.0;
   DATA[105,10] := 2.0;
   DATA[105,11] := 19.59793;
   DATA[105,12] := 2.209525;
   DATA[105,13] := 960.3307;
   DATA[105,14] := 1.0;
   DATA[105,15] := 2.0;
   DATA[105,16] := 1.0;
   DATA[105,17] := 1.0;
   DATA[105,18] := 1.0;
   DATA[105,19] := 2.0;
   DATA[105,20] := 148.808;
   DATA[105,21] := 156.1907;
   DATA[105,22] := 1.718515;
   DATA[105,23] := 952.7557;
   DATA[105,24] := 2.0;
   DATA[105,25] := 2.0;
   DATA[105,26] := 7.877019;
   DATA[105,27] := 145.0397;
   DATA[105,28] := 264.2592;
   DATA[105,29] := 12.07383;
   DATA[105,30] := 1.725583;
   DATA[105,31] := 1.256052;
   DATA[105,32] := 0.7353967;
   DATA[105,33] := 0.3086186;
   DATA[105,34] := 2.0;
   DATA[105,35] := 251.0414;
   DATA[105,36] := 1.649953;
   DATA[105,37] := 189.8071;
   DATA[105,38] := 0.000128152;
   DATA[105,39] := 1.0;
   DATA[106,0] := 2.444992;
   DATA[106,1] := 523.4748;
   DATA[106,2] := 2.0;
   DATA[106,3] := 2.0;
   DATA[106,4] := 262.1764;
   DATA[106,5] := 8.39163;
   DATA[106,6] := 328.4286;
   DATA[106,7] := 2.445263;
   DATA[106,8] := 2.0;
   DATA[106,9] := 2.0;
   DATA[106,10] := 2.0;
   DATA[106,11] := 19.65555;
   DATA[106,12] := 2.209525;
   DATA[106,13] := 960.3708;
   DATA[106,14] := 1.0;
   DATA[106,15] := 2.0;
   DATA[106,16] := 1.0;
   DATA[106,17] := 1.0;
   DATA[106,18] := 1.0;
   DATA[106,19] := 2.0;
   DATA[106,20] := 148.808;
   DATA[106,21] := 156.1907;
   DATA[106,22] := 1.719156;
   DATA[106,23] := 952.6403;
   DATA[106,24] := 2.0;
   DATA[106,25] := 2.0;
   DATA[106,26] := 7.877019;
   DATA[106,27] := 145.0397;
   DATA[106,28] := 264.2592;
   DATA[106,29] := 12.07383;
   DATA[106,30] := 1.726737;
   DATA[106,31] := 1.269502;
   DATA[106,32] := 0.7353967;
   DATA[106,33] := 0.3086186;
   DATA[106,34] := 2.0;
   DATA[106,35] := 251.0414;
   DATA[106,36] := 1.649953;
   DATA[106,37] := 189.8071;
   DATA[106,38] := 0.000128152;
   DATA[106,39] := 1.0;
   DATA[107,0] := 2.492714;
   DATA[107,1] := 523.3177;
   DATA[107,2] := 2.0;
   DATA[107,3] := 2.0;
   DATA[107,4] := 262.1764;
   DATA[107,5] := 8.39163;
   DATA[107,6] := 328.4286;
   DATA[107,7] := 2.44616;
   DATA[107,8] := 2.0;
   DATA[107,9] := 2.0;
   DATA[107,10] := 2.0;
   DATA[107,11] := 19.69076;
   DATA[107,12] := 2.211447;
   DATA[107,13] := 959.8901;
   DATA[107,14] := 1.0;
   DATA[107,15] := 2.0;
   DATA[107,16] := 1.0;
   DATA[107,17] := 1.0;
   DATA[107,18] := 1.0;
   DATA[107,19] := 2.0;
   DATA[107,20] := 148.808;
   DATA[107,21] := 156.1907;
   DATA[107,22] := 1.719156;
   DATA[107,23] := 953.1402;
   DATA[107,24] := 2.0;
   DATA[107,25] := 2.0;
   DATA[107,26] := 7.877019;
   DATA[107,27] := 145.0397;
   DATA[107,28] := 264.2592;
   DATA[107,29] := 12.07383;
   DATA[107,30] := 1.726993;
   DATA[107,31] := 1.272064;
   DATA[107,32] := 0.7353967;
   DATA[107,33] := 0.3086186;
   DATA[107,34] := 2.0;
   DATA[107,35] := 251.0414;
   DATA[107,36] := 1.826162;
   DATA[107,37] := 189.8071;
   DATA[107,38] := 0.000128152;
   DATA[107,39] := 1.0;
   DATA[108,0] := 2.533709;
   DATA[108,1] := 523.4355;
   DATA[108,2] := 2.0;
   DATA[108,3] := 2.0;
   DATA[108,4] := 262.1764;
   DATA[108,5] := 8.39163;
   DATA[108,6] := 328.4286;
   DATA[108,7] := 2.44616;
   DATA[108,8] := 2.0;
   DATA[108,9] := 2.0;
   DATA[108,10] := 2.0;
   DATA[108,11] := 19.69076;
   DATA[108,12] := 2.211447;
   DATA[108,13] := 959.8901;
   DATA[108,14] := 1.0;
   DATA[108,15] := 2.0;
   DATA[108,16] := 1.0;
   DATA[108,17] := 1.0;
   DATA[108,18] := 1.0;
   DATA[108,19] := 2.0;
   DATA[108,20] := 148.808;
   DATA[108,21] := 156.1907;
   DATA[108,22] := 1.716849;
   DATA[108,23] := 953.0248;
   DATA[108,24] := 2.0;
   DATA[108,25] := 2.0;
   DATA[108,26] := 7.877019;
   DATA[108,27] := 145.0397;
   DATA[108,28] := 264.2592;
   DATA[108,29] := 12.07383;
   DATA[108,30] := 1.726993;
   DATA[108,31] := 1.278596;
   DATA[108,32] := 0.7353967;
   DATA[108,33] := 0.3086186;
   DATA[108,34] := 2.0;
   DATA[108,35] := 251.0414;
   DATA[108,36] := 1.665972;
   DATA[108,37] := 189.8071;
   DATA[108,38] := 0.000128152;
   DATA[108,39] := 1.0;
   DATA[109,0] := 2.574064;
   DATA[109,1] := 523.0823;
   DATA[109,2] := 2.0;
   DATA[109,3] := 2.0;
   DATA[109,4] := 262.1764;
   DATA[109,5] := 8.39163;
   DATA[109,6] := 328.4286;
   DATA[109,7] := 2.44616;
   DATA[109,8] := 2.0;
   DATA[109,9] := 2.0;
   DATA[109,10] := 2.0;
   DATA[109,11] := 19.69076;
   DATA[109,12] := 2.211447;
   DATA[109,13] := 960.1304;
   DATA[109,14] := 1.0;
   DATA[109,15] := 2.0;
   DATA[109,16] := 1.0;
   DATA[109,17] := 1.0;
   DATA[109,18] := 1.0;
   DATA[109,19] := 2.0;
   DATA[109,20] := 148.808;
   DATA[109,21] := 156.1907;
   DATA[109,22] := 1.716592;
   DATA[109,23] := 953.0633;
   DATA[109,24] := 2.0;
   DATA[109,25] := 2.0;
   DATA[109,26] := 7.877019;
   DATA[109,27] := 145.0397;
   DATA[109,28] := 264.2592;
   DATA[109,29] := 12.07383;
   DATA[109,30] := 1.726993;
   DATA[109,31] := 1.281542;
   DATA[109,32] := 0.7353967;
   DATA[109,33] := 0.3086186;
   DATA[109,34] := 2.0;
   DATA[109,35] := 250.9773;
   DATA[109,36] := 1.665972;
   DATA[109,37] := 189.5347;
   DATA[109,38] := 0.000128152;
   DATA[109,39] := 1.0;
   DATA[110,0] := 2.602569;
   DATA[110,1] := 523.1608;
   DATA[110,2] := 2.0;
   DATA[110,3] := 2.0;
   DATA[110,4] := 262.1764;
   DATA[110,5] := 8.39163;
   DATA[110,6] := 328.4286;
   DATA[110,7] := 2.444623;
   DATA[110,8] := 2.0;
   DATA[110,9] := 2.0;
   DATA[110,10] := 2.0;
   DATA[110,11] := 19.69076;
   DATA[110,12] := 2.209653;
   DATA[110,13] := 960.1304;
   DATA[110,14] := 1.0;
   DATA[110,15] := 2.0;
   DATA[110,16] := 1.0;
   DATA[110,17] := 1.0;
   DATA[110,18] := 1.0;
   DATA[110,19] := 2.0;
   DATA[110,20] := 148.808;
   DATA[110,21] := 156.1907;
   DATA[110,22] := 1.715567;
   DATA[110,23] := 953.2171;
   DATA[110,24] := 2.0;
   DATA[110,25] := 2.0;
   DATA[110,26] := 7.877019;
   DATA[110,27] := 145.0397;
   DATA[110,28] := 264.2592;
   DATA[110,29] := 12.07383;
   DATA[110,30] := 1.726993;
   DATA[110,31] := 1.276675;
   DATA[110,32] := 0.7353967;
   DATA[110,33] := 0.3070813;
   DATA[110,34] := 2.0;
   DATA[110,35] := 250.8171;
   DATA[110,36] := 1.665972;
   DATA[110,37] := 189.5347;
   DATA[110,38] := 0.000128152;
   DATA[110,39] := 1.0;
   DATA[111,0] := 2.637158;
   DATA[111,1] := 523.2393;
   DATA[111,2] := 2.0;
   DATA[111,3] := 2.0;
   DATA[111,4] := 262.1764;
   DATA[111,5] := 8.39163;
   DATA[111,6] := 328.4286;
   DATA[111,7] := 2.444623;
   DATA[111,8] := 2.0;
   DATA[111,9] := 2.0;
   DATA[111,10] := 2.0;
   DATA[111,11] := 19.73238;
   DATA[111,12] := 2.209525;
   DATA[111,13] := 959.7299;
   DATA[111,14] := 1.0;
   DATA[111,15] := 2.0;
   DATA[111,16] := 1.0;
   DATA[111,17] := 1.0;
   DATA[111,18] := 1.0;
   DATA[111,19] := 2.0;
   DATA[111,20] := 148.808;
   DATA[111,21] := 156.1907;
   DATA[111,22] := 1.715567;
   DATA[111,23] := 953.1402;
   DATA[111,24] := 2.0;
   DATA[111,25] := 2.0;
   DATA[111,26] := 7.877019;
   DATA[111,27] := 145.0397;
   DATA[111,28] := 264.2592;
   DATA[111,29] := 12.07383;
   DATA[111,30] := 1.726993;
   DATA[111,31] := 1.290509;
   DATA[111,32] := 0.7353967;
   DATA[111,33] := 0.3068251;
   DATA[111,34] := 2.0;
   DATA[111,35] := 250.8171;
   DATA[111,36] := 1.665972;
   DATA[111,37] := 189.5347;
   DATA[111,38] := 0.000128152;
   DATA[111,39] := 1.0;
   DATA[112,0] := 2.654774;
   DATA[112,1] := 523.514;
   DATA[112,2] := 2.0;
   DATA[112,3] := 2.0;
   DATA[112,4] := 262.1443;
   DATA[112,5] := 8.39163;
   DATA[112,6] := 328.4286;
   DATA[112,7] := 2.441803;
   DATA[112,8] := 2.0;
   DATA[112,9] := 2.0;
   DATA[112,10] := 2.0;
   DATA[112,11] := 19.74838;
   DATA[112,12] := 2.209525;
   DATA[112,13] := 959.6097;
   DATA[112,14] := 1.0;
   DATA[112,15] := 2.0;
   DATA[112,16] := 1.0;
   DATA[112,17] := 1.0;
   DATA[112,18] := 1.0;
   DATA[112,19] := 2.0;
   DATA[112,20] := 148.808;
   DATA[112,21] := 156.1907;
   DATA[112,22] := 1.715567;
   DATA[112,23] := 953.4094;
   DATA[112,24] := 2.0;
   DATA[112,25] := 2.0;
   DATA[112,26] := 7.877019;
   DATA[112,27] := 145.0397;
   DATA[112,28] := 264.2592;
   DATA[112,29] := 12.07383;
   DATA[112,30] := 1.726993;
   DATA[112,31] := 1.290765;
   DATA[112,32] := 0.7353967;
   DATA[112,33] := 0.3068251;
   DATA[112,34] := 2.0;
   DATA[112,35] := 250.8171;
   DATA[112,36] := 1.665972;
   DATA[112,37] := 189.6949;
   DATA[112,38] := 0.000128152;
   DATA[112,39] := 1.0;
   DATA[113,0] := 2.66214;
   DATA[113,1] := 523.8673;
   DATA[113,2] := 2.0;
   DATA[113,3] := 2.0;
   DATA[113,4] := 262.1443;
   DATA[113,5] := 8.39163;
   DATA[113,6] := 328.4286;
   DATA[113,7] := 2.439625;
   DATA[113,8] := 2.0;
   DATA[113,9] := 2.0;
   DATA[113,10] := 2.0;
   DATA[113,11] := 19.74838;
   DATA[113,12] := 2.210166;
   DATA[113,13] := 959.7299;
   DATA[113,14] := 1.0;
   DATA[113,15] := 2.0;
   DATA[113,16] := 1.0;
   DATA[113,17] := 1.0;
   DATA[113,18] := 1.0;
   DATA[113,19] := 2.0;
   DATA[113,20] := 148.808;
   DATA[113,21] := 156.1907;
   DATA[113,22] := 1.715567;
   DATA[113,23] := 953.5247;
   DATA[113,24] := 2.0;
   DATA[113,25] := 2.0;
   DATA[113,26] := 7.877019;
   DATA[113,27] := 145.0397;
   DATA[113,28] := 264.2592;
   DATA[113,29] := 12.07383;
   DATA[113,30] := 1.726993;
   DATA[113,31] := 1.286025;
   DATA[113,32] := 0.7353967;
   DATA[113,33] := 0.3068251;
   DATA[113,34] := 2.0;
   DATA[113,35] := 250.8171;
   DATA[113,36] := 1.665972;
   DATA[113,37] := 189.6949;
   DATA[113,38] := 0.000128152;
   DATA[113,39] := 1.0;
   DATA[114,0] := 2.647407;
   DATA[114,1] := 524.2206;
   DATA[114,2] := 2.0;
   DATA[114,3] := 2.0;
   DATA[114,4] := 262.1443;
   DATA[114,5] := 8.39163;
   DATA[114,6] := 328.4286;
   DATA[114,7] := 2.43924;
   DATA[114,8] := 2.0;
   DATA[114,9] := 2.0;
   DATA[114,10] := 2.0;
   DATA[114,11] := 19.74838;
   DATA[114,12] := 2.210166;
   DATA[114,13] := 959.5697;
   DATA[114,14] := 1.0;
   DATA[114,15] := 2.0;
   DATA[114,16] := 1.0;
   DATA[114,17] := 1.0;
   DATA[114,18] := 1.0;
   DATA[114,19] := 2.0;
   DATA[114,20] := 148.808;
   DATA[114,21] := 156.1907;
   DATA[114,22] := 1.715567;
   DATA[114,23] := 953.5247;
   DATA[114,24] := 2.0;
   DATA[114,25] := 2.0;
   DATA[114,26] := 7.877019;
   DATA[114,27] := 145.0397;
   DATA[114,28] := 264.2592;
   DATA[114,29] := 12.07383;
   DATA[114,30] := 1.726993;
   DATA[114,31] := 1.286794;
   DATA[114,32] := 0.7353967;
   DATA[114,33] := 0.3068251;
   DATA[114,34] := 2.0;
   DATA[114,35] := 250.8171;
   DATA[114,36] := 1.665972;
   DATA[114,37] := 189.6949;
   DATA[114,38] := 0.000128152;
   DATA[114,39] := 1.0;
   DATA[115,0] := 2.630433;
   DATA[115,1] := 524.2206;
   DATA[115,2] := 2.0;
   DATA[115,3] := 2.0;
   DATA[115,4] := 262.1443;
   DATA[115,5] := 8.39163;
   DATA[115,6] := 328.4286;
   DATA[115,7] := 2.43924;
   DATA[115,8] := 2.0;
   DATA[115,9] := 2.0;
   DATA[115,10] := 2.0;
   DATA[115,11] := 19.70037;
   DATA[115,12] := 2.210166;
   DATA[115,13] := 959.77;
   DATA[115,14] := 1.0;
   DATA[115,15] := 2.0;
   DATA[115,16] := 1.0;
   DATA[115,17] := 1.0;
   DATA[115,18] := 1.0;
   DATA[115,19] := 2.0;
   DATA[115,20] := 148.808;
   DATA[115,21] := 156.1907;
   DATA[115,22] := 1.715567;
   DATA[115,23] := 953.717;
   DATA[115,24] := 2.0;
   DATA[115,25] := 2.0;
   DATA[115,26] := 7.877019;
   DATA[115,27] := 145.0397;
   DATA[115,28] := 264.2592;
   DATA[115,29] := 12.07383;
   DATA[115,30] := 1.726993;
   DATA[115,31] := 1.272576;
   DATA[115,32] := 0.7353967;
   DATA[115,33] := 0.3068251;
   DATA[115,34] := 2.0;
   DATA[115,35] := 250.9453;
   DATA[115,36] := 1.665972;
   DATA[115,37] := 189.6949;
   DATA[115,38] := 0.000128152;
   DATA[115,39] := 1.0;
   DATA[116,0] := 2.622426;
   DATA[116,1] := 524.0636;
   DATA[116,2] := 2.0;
   DATA[116,3] := 2.0;
   DATA[116,4] := 262.1443;
   DATA[116,5] := 8.39163;
   DATA[116,6] := 328.4286;
   DATA[116,7] := 2.441803;
   DATA[116,8] := 2.0;
   DATA[116,9] := 2.0;
   DATA[116,10] := 2.0;
   DATA[116,11] := 19.65555;
   DATA[116,12] := 2.212215;
   DATA[116,13] := 960.2106;
   DATA[116,14] := 1.0;
   DATA[116,15] := 2.0;
   DATA[116,16] := 1.0;
   DATA[116,17] := 1.0;
   DATA[116,18] := 1.0;
   DATA[116,19] := 2.0;
   DATA[116,20] := 148.808;
   DATA[116,21] := 156.1907;
   DATA[116,22] := 1.716208;
   DATA[116,23] := 953.9861;
   DATA[116,24] := 2.0;
   DATA[116,25] := 2.0;
   DATA[116,26] := 7.877019;
   DATA[116,27] := 145.0397;
   DATA[116,28] := 264.2592;
   DATA[116,29] := 12.07383;
   DATA[116,30] := 1.726993;
   DATA[116,31] := 1.272576;
   DATA[116,32] := 0.7353967;
   DATA[116,33] := 0.3068251;
   DATA[116,34] := 2.0;
   DATA[116,35] := 250.9453;
   DATA[116,36] := 1.665972;
   DATA[116,37] := 189.6949;
   DATA[116,38] := 0.000128152;
   DATA[116,39] := 1.0;
   DATA[117,0] := 2.620184;
   DATA[117,1] := 523.9458;
   DATA[117,2] := 2.0;
   DATA[117,3] := 2.0;
   DATA[117,4] := 262.1443;
   DATA[117,5] := 8.39163;
   DATA[117,6] := 328.4286;
   DATA[117,7] := 2.441803;
   DATA[117,8] := 2.0;
   DATA[117,9] := 2.0;
   DATA[117,10] := 2.0;
   DATA[117,11] := 19.65555;
   DATA[117,12] := 2.212215;
   DATA[117,13] := 960.4108;
   DATA[117,14] := 1.0;
   DATA[117,15] := 2.0;
   DATA[117,16] := 1.0;
   DATA[117,17] := 1.0;
   DATA[117,18] := 1.0;
   DATA[117,19] := 2.0;
   DATA[117,20] := 148.808;
   DATA[117,21] := 156.1907;
   DATA[117,22] := 1.716849;
   DATA[117,23] := 954.14;
   DATA[117,24] := 2.0;
   DATA[117,25] := 2.0;
   DATA[117,26] := 7.877019;
   DATA[117,27] := 145.0397;
   DATA[117,28] := 264.2592;
   DATA[117,29] := 12.07383;
   DATA[117,30] := 1.726993;
   DATA[117,31] := 1.276675;
   DATA[117,32] := 0.7353967;
   DATA[117,33] := 0.3081703;
   DATA[117,34] := 2.0;
   DATA[117,35] := 250.9453;
   DATA[117,36] := 1.665972;
   DATA[117,37] := 189.6949;
   DATA[117,38] := 0.000128152;
   DATA[117,39] := 1.0;
   DATA[118,0] := 2.608013;
   DATA[118,1] := 523.4748;
   DATA[118,2] := 2.0;
   DATA[118,3] := 2.0;
   DATA[118,4] := 262.1443;
   DATA[118,5] := 8.39163;
   DATA[118,6] := 328.4286;
   DATA[118,7] := 2.440137;
   DATA[118,8] := 2.0;
   DATA[118,9] := 2.0;
   DATA[118,10] := 2.0;
   DATA[118,11] := 19.65555;
   DATA[118,12] := 2.212215;
   DATA[118,13] := 960.6111;
   DATA[118,14] := 1.0;
   DATA[118,15] := 2.0;
   DATA[118,16] := 1.0;
   DATA[118,17] := 1.0;
   DATA[118,18] := 1.0;
   DATA[118,19] := 2.0;
   DATA[118,20] := 148.808;
   DATA[118,21] := 156.1907;
   DATA[118,22] := 1.716849;
   DATA[118,23] := 953.9861;
   DATA[118,24] := 2.0;
   DATA[118,25] := 2.0;
   DATA[118,26] := 7.877019;
   DATA[118,27] := 145.091;
   DATA[118,28] := 264.2592;
   DATA[118,29] := 12.07383;
   DATA[118,30] := 1.725327;
   DATA[118,31] := 1.276034;
   DATA[118,32] := 0.7353967;
   DATA[118,33] := 0.3084265;
   DATA[118,34] := 2.0;
   DATA[118,35] := 250.9453;
   DATA[118,36] := 1.665972;
   DATA[118,37] := 189.6949;
   DATA[118,38] := 0.000128152;
   DATA[118,39] := 1.0;
   DATA[119,0] := 2.586875;
   DATA[119,1] := 523.5533;
   DATA[119,2] := 2.0;
   DATA[119,3] := 2.0;
   DATA[119,4] := 262.1443;
   DATA[119,5] := 8.39163;
   DATA[119,6] := 328.4286;
   DATA[119,7] := 2.440137;
   DATA[119,8] := 2.0;
   DATA[119,9] := 2.0;
   DATA[119,10] := 2.0;
   DATA[119,11] := 19.65555;
   DATA[119,12] := 2.2126;
   DATA[119,13] := 961.0116;
   DATA[119,14] := 1.0;
   DATA[119,15] := 2.0;
   DATA[119,16] := 1.0;
   DATA[119,17] := 1.0;
   DATA[119,18] := 1.0;
   DATA[119,19] := 2.0;
   DATA[119,20] := 148.808;
   DATA[119,21] := 156.0625;
   DATA[119,22] := 1.716849;
   DATA[119,23] := 954.1015;
   DATA[119,24] := 2.0;
   DATA[119,25] := 2.0;
   DATA[119,26] := 7.877019;
   DATA[119,27] := 145.091;
   DATA[119,28] := 264.131;
   DATA[119,29] := 12.07383;
   DATA[119,30] := 1.725327;
   DATA[119,31] := 1.283079;
   DATA[119,32] := 0.7353967;
   DATA[119,33] := 0.3084265;
   DATA[119,34] := 2.0;
   DATA[119,35] := 250.9453;
   DATA[119,36] := 1.665972;
   DATA[119,37] := 189.6949;
   DATA[119,38] := 0.000128152;
   DATA[119,39] := 1.0;
   DATA[120,0] := 2.574064;
   DATA[120,1] := 523.8281;
   DATA[120,2] := 2.0;
   DATA[120,3] := 2.0;
   DATA[120,4] := 262.1443;
   DATA[120,5] := 8.39163;
   DATA[120,6] := 328.4286;
   DATA[120,7] := 2.440137;
   DATA[120,8] := 2.0;
   DATA[120,9] := 2.0;
   DATA[120,10] := 2.0;
   DATA[120,11] := 19.63954;
   DATA[120,12] := 2.2126;
   DATA[120,13] := 960.8113;
   DATA[120,14] := 1.0;
   DATA[120,15] := 2.0;
   DATA[120,16] := 1.0;
   DATA[120,17] := 1.0;
   DATA[120,18] := 1.0;
   DATA[120,19] := 2.0;
   DATA[120,20] := 148.808;
   DATA[120,21] := 156.0625;
   DATA[120,22] := 1.715824;
   DATA[120,23] := 954.3707;
   DATA[120,24] := 2.0;
   DATA[120,25] := 2.0;
   DATA[120,26] := 7.877019;
   DATA[120,27] := 145.091;
   DATA[120,28] := 264.0669;
   DATA[120,29] := 12.07383;
   DATA[120,30] := 1.725327;
   DATA[120,31] := 1.283079;
   DATA[120,32] := 0.7353967;
   DATA[120,33] := 0.3084265;
   DATA[120,34] := 2.0;
   DATA[120,35] := 250.9453;
   DATA[120,36] := 1.665972;
   DATA[120,37] := 189.6949;
   DATA[120,38] := 0.000128152;
   DATA[120,39] := 1.0;
   DATA[121,0] := 2.560292;
   DATA[121,1] := 523.7496;
   DATA[121,2] := 2.0;
   DATA[121,3] := 2.0;
   DATA[121,4] := 262.1443;
   DATA[121,5] := 8.39163;
   DATA[121,6] := 328.4286;
   DATA[121,7] := 2.440137;
   DATA[121,8] := 2.0;
   DATA[121,9] := 2.0;
   DATA[121,10] := 2.0;
   DATA[121,11] := 19.62033;
   DATA[121,12] := 2.2126;
   DATA[121,13] := 960.8113;
   DATA[121,14] := 1.0;
   DATA[121,15] := 2.0;
   DATA[121,16] := 1.0;
   DATA[121,17] := 1.0;
   DATA[121,18] := 1.0;
   DATA[121,19] := 2.0;
   DATA[121,20] := 148.808;
   DATA[121,21] := 156.0625;
   DATA[121,22] := 1.715824;
   DATA[121,23] := 955.0628;
   DATA[121,24] := 2.0;
   DATA[121,25] := 2.0;
   DATA[121,26] := 7.877019;
   DATA[121,27] := 145.091;
   DATA[121,28] := 264.0669;
   DATA[121,29] := 12.07383;
   DATA[121,30] := 1.725327;
   DATA[121,31] := 1.283079;
   DATA[121,32] := 0.7353967;
   DATA[121,33] := 0.3084265;
   DATA[121,34] := 2.0;
   DATA[121,35] := 250.9453;
   DATA[121,36] := 1.665972;
   DATA[121,37] := 189.6949;
   DATA[121,38] := 0.000128152;
   DATA[121,39] := 1.0;
   DATA[122,0] := 2.541716;
   DATA[122,1] := 524.0636;
   DATA[122,2] := 2.0;
   DATA[122,3] := 2.0;
   DATA[122,4] := 262.1443;
   DATA[122,5] := 8.39163;
   DATA[122,6] := 328.4286;
   DATA[122,7] := 2.440137;
   DATA[122,8] := 2.0;
   DATA[122,9] := 2.0;
   DATA[122,10] := 2.0;
   DATA[122,11] := 19.62033;
   DATA[122,12] := 2.2126;
   DATA[122,13] := 960.7713;
   DATA[122,14] := 1.0;
   DATA[122,15] := 2.0;
   DATA[122,16] := 1.0;
   DATA[122,17] := 1.0;
   DATA[122,18] := 1.0;
   DATA[122,19] := 2.0;
   DATA[122,20] := 148.808;
   DATA[122,21] := 156.0625;
   DATA[122,22] := 1.715824;
   DATA[122,23] := 955.0628;
   DATA[122,24] := 2.0;
   DATA[122,25] := 2.0;
   DATA[122,26] := 7.877019;
   DATA[122,27] := 145.091;
   DATA[122,28] := 264.0669;
   DATA[122,29] := 12.07383;
   DATA[122,30] := 1.725327;
   DATA[122,31] := 1.292046;
   DATA[122,32] := 0.7353967;
   DATA[122,33] := 0.3084265;
   DATA[122,34] := 2.0;
   DATA[122,35] := 250.9453;
   DATA[122,36] := 1.665972;
   DATA[122,37] := 189.6949;
   DATA[122,38] := 0.000128152;
   DATA[122,39] := 1.0;
   DATA[123,0] := 2.520898;
   DATA[123,1] := 524.5346;
   DATA[123,2] := 2.0;
   DATA[123,3] := 2.0;
   DATA[123,4] := 262.1443;
   DATA[123,5] := 8.39163;
   DATA[123,6] := 328.4286;
   DATA[123,7] := 2.440137;
   DATA[123,8] := 2.0;
   DATA[123,9] := 2.0;
   DATA[123,10] := 2.0;
   DATA[123,11] := 19.67796;
   DATA[123,12] := 2.2126;
   DATA[123,13] := 960.6111;
   DATA[123,14] := 1.0;
   DATA[123,15] := 2.0;
   DATA[123,16] := 1.0;
   DATA[123,17] := 1.0;
   DATA[123,18] := 1.0;
   DATA[123,19] := 2.0;
   DATA[123,20] := 148.808;
   DATA[123,21] := 156.0625;
   DATA[123,22] := 1.715824;
   DATA[123,23] := 954.9474;
   DATA[123,24] := 2.0;
   DATA[123,25] := 2.0;
   DATA[123,26] := 7.877019;
   DATA[123,27] := 145.091;
   DATA[123,28] := 264.0989;
   DATA[123,29] := 12.26609;
   DATA[123,30] := 1.725327;
   DATA[123,31] := 1.297554;
   DATA[123,32] := 0.7353967;
   DATA[123,33] := 0.3084265;
   DATA[123,34] := 2.0;
   DATA[123,35] := 250.9453;
   DATA[123,36] := 1.665972;
   DATA[123,37] := 189.6949;
   DATA[123,38] := 0.000128152;
   DATA[123,39] := 1.0;
   DATA[124,0] := 2.509688;
   DATA[124,1] := 524.5346;
   DATA[124,2] := 2.0;
   DATA[124,3] := 2.0;
   DATA[124,4] := 262.1443;
   DATA[124,5] := 8.39163;
   DATA[124,6] := 328.4286;
   DATA[124,7] := 2.440137;
   DATA[124,8] := 2.0;
   DATA[124,9] := 2.0;
   DATA[124,10] := 2.0;
   DATA[124,11] := 19.67796;
   DATA[124,12] := 2.2126;
   DATA[124,13] := 960.571;
   DATA[124,14] := 1.0;
   DATA[124,15] := 2.0;
   DATA[124,16] := 1.0;
   DATA[124,17] := 1.0;
   DATA[124,18] := 1.0;
   DATA[124,19] := 2.0;
   DATA[124,20] := 148.808;
   DATA[124,21] := 156.0625;
   DATA[124,22] := 1.715824;
   DATA[124,23] := 954.9474;
   DATA[124,24] := 2.0;
   DATA[124,25] := 2.0;
   DATA[124,26] := 7.877019;
   DATA[124,27] := 145.091;
   DATA[124,28] := 264.2912;
   DATA[124,29] := 12.26609;
   DATA[124,30] := 1.725327;
   DATA[124,31] := 1.302037;
   DATA[124,32] := 0.7353967;
   DATA[124,33] := 0.3084265;
   DATA[124,34] := 2.0;
   DATA[124,35] := 250.9453;
   DATA[124,36] := 1.665972;
   DATA[124,37] := 189.6949;
   DATA[124,38] := 0.000128152;
   DATA[124,39] := 1.0;
   DATA[125,0] := 2.487269;
   DATA[125,1] := 525.0056;
   DATA[125,2] := 2.0;
   DATA[125,3] := 2.0;
   DATA[125,4] := 262.1443;
   DATA[125,5] := 8.39163;
   DATA[125,6] := 328.4286;
   DATA[125,7] := 2.440137;
   DATA[125,8] := 2.0;
   DATA[125,9] := 2.0;
   DATA[125,10] := 2.0;
   DATA[125,11] := 19.67796;
   DATA[125,12] := 2.2126;
   DATA[125,13] := 960.6511;
   DATA[125,14] := 1.0;
   DATA[125,15] := 2.0;
   DATA[125,16] := 1.0;
   DATA[125,17] := 1.0;
   DATA[125,18] := 1.0;
   DATA[125,19] := 2.0;
   DATA[125,20] := 148.808;
   DATA[125,21] := 155.9856;
   DATA[125,22] := 1.715824;
   DATA[125,23] := 955.3704;
   DATA[125,24] := 2.0;
   DATA[125,25] := 2.0;
   DATA[125,26] := 7.877019;
   DATA[125,27] := 145.091;
   DATA[125,28] := 264.2912;
   DATA[125,29] := 12.26609;
   DATA[125,30] := 1.725327;
   DATA[125,31] := 1.302037;
   DATA[125,32] := 0.7353967;
   DATA[125,33] := 0.3084265;
   DATA[125,34] := 2.0;
   DATA[125,35] := 250.9453;
   DATA[125,36] := 1.665972;
   DATA[125,37] := 189.6949;
   DATA[125,38] := 0.000128152;
   DATA[125,39] := 1.0;
   DATA[126,0] := 2.46581;
   DATA[126,1] := 525.5944;
   DATA[126,2] := 2.0;
   DATA[126,3] := 2.0;
   DATA[126,4] := 262.1443;
   DATA[126,5] := 8.39163;
   DATA[126,6] := 328.4286;
   DATA[126,7] := 2.440137;
   DATA[126,8] := 2.0;
   DATA[126,9] := 2.0;
   DATA[126,10] := 2.0;
   DATA[126,11] := 19.74198;
   DATA[126,12] := 2.2126;
   DATA[126,13] := 961.0517;
   DATA[126,14] := 1.0;
   DATA[126,15] := 2.0;
   DATA[126,16] := 1.0;
   DATA[126,17] := 1.0;
   DATA[126,18] := 1.0;
   DATA[126,19] := 2.0;
   DATA[126,20] := 148.808;
   DATA[126,21] := 155.8575;
   DATA[126,22] := 1.715824;
   DATA[126,23] := 955.6396;
   DATA[126,24] := 2.0;
   DATA[126,25] := 2.0;
   DATA[126,26] := 7.877019;
   DATA[126,27] := 145.091;
   DATA[126,28] := 264.2912;
   DATA[126,29] := 12.26609;
   DATA[126,30] := 1.725327;
   DATA[126,31] := 1.286025;
   DATA[126,32] := 0.7353967;
   DATA[126,33] := 0.3084265;
   DATA[126,34] := 2.0;
   DATA[126,35] := 250.9453;
   DATA[126,36] := 1.665972;
   DATA[126,37] := 189.6949;
   DATA[126,38] := 0.000128152;
   DATA[126,39] := 1.0;
   DATA[127,0] := 2.455241;
   DATA[127,1] := 525.9084;
   DATA[127,2] := 2.0;
   DATA[127,3] := 2.0;
   DATA[127,4] := 262.1443;
   DATA[127,5] := 8.39163;
   DATA[127,6] := 328.4286;
   DATA[127,7] := 2.440137;
   DATA[127,8] := 2.0;
   DATA[127,9] := 2.0;
   DATA[127,10] := 2.0;
   DATA[127,11] := 19.74198;
   DATA[127,12] := 2.2126;
   DATA[127,13] := 960.9716;
   DATA[127,14] := 1.0;
   DATA[127,15] := 2.0;
   DATA[127,16] := 1.0;
   DATA[127,17] := 1.0;
   DATA[127,18] := 1.0;
   DATA[127,19] := 2.0;
   DATA[127,20] := 148.808;
   DATA[127,21] := 155.8575;
   DATA[127,22] := 1.715824;
   DATA[127,23] := 955.7165;
   DATA[127,24] := 2.0;
   DATA[127,25] := 2.0;
   DATA[127,26] := 7.877019;
   DATA[127,27] := 145.091;
   DATA[127,28] := 264.2912;
   DATA[127,29] := 12.26609;
   DATA[127,30] := 1.725327;
   DATA[127,31] := 1.272192;
   DATA[127,32] := 0.7353967;
   DATA[127,33] := 0.3066329;
   DATA[127,34] := 2.0;
   DATA[127,35] := 250.9453;
   DATA[127,36] := 1.665972;
   DATA[127,37] := 189.6949;
   DATA[127,38] := 0.000128152;
   DATA[127,39] := 1.0;
   DATA[128,0] := 2.439868;
   DATA[128,1] := 525.9869;
   DATA[128,2] := 2.0;
   DATA[128,3] := 2.0;
   DATA[128,4] := 262.1443;
   DATA[128,5] := 8.39163;
   DATA[128,6] := 328.4286;
   DATA[128,7] := 2.440137;
   DATA[128,8] := 2.0;
   DATA[128,9] := 2.0;
   DATA[128,10] := 2.0;
   DATA[128,11] := 19.74198;
   DATA[128,12] := 2.2126;
   DATA[128,13] := 961.2119;
   DATA[128,14] := 1.0;
   DATA[128,15] := 2.0;
   DATA[128,16] := 1.0;
   DATA[128,17] := 1.0;
   DATA[128,18] := 1.0;
   DATA[128,19] := 2.0;
   DATA[128,20] := 148.808;
   DATA[128,21] := 155.8575;
   DATA[128,22] := 1.715824;
   DATA[128,23] := 955.6396;
   DATA[128,24] := 2.0;
   DATA[128,25] := 2.0;
   DATA[128,26] := 7.877019;
   DATA[128,27] := 145.1423;
   DATA[128,28] := 264.2912;
   DATA[128,29] := 12.07383;
   DATA[128,30] := 1.725327;
   DATA[128,31] := 1.261432;
   DATA[128,32] := 0.7353967;
   DATA[128,33] := 0.3066329;
   DATA[128,34] := 2.0;
   DATA[128,35] := 250.9453;
   DATA[128,36] := 1.665972;
   DATA[128,37] := 189.6949;
   DATA[128,38] := 0.000128152;
   DATA[128,39] := 1.0;
   DATA[129,0] := 2.428338;
   DATA[129,1] := 526.0655;
   DATA[129,2] := 2.0;
   DATA[129,3] := 2.0;
   DATA[129,4] := 262.1443;
   DATA[129,5] := 8.39163;
   DATA[129,6] := 328.4286;
   DATA[129,7] := 2.440137;
   DATA[129,8] := 2.0;
   DATA[129,9] := 2.0;
   DATA[129,10] := 2.0;
   DATA[129,11] := 19.74198;
   DATA[129,12] := 2.210294;
   DATA[129,13] := 961.1318;
   DATA[129,14] := 1.0;
   DATA[129,15] := 2.0;
   DATA[129,16] := 1.0;
   DATA[129,17] := 1.0;
   DATA[129,18] := 1.0;
   DATA[129,19] := 2.0;
   DATA[129,20] := 148.808;
   DATA[129,21] := 155.7806;
   DATA[129,22] := 1.715824;
   DATA[129,23] := 955.8318;
   DATA[129,24] := 2.0;
   DATA[129,25] := 2.0;
   DATA[129,26] := 7.877019;
   DATA[129,27] := 145.1423;
   DATA[129,28] := 264.2912;
   DATA[129,29] := 12.07383;
   DATA[129,30] := 1.725327;
   DATA[129,31] := 1.267452;
   DATA[129,32] := 0.7353967;
   DATA[129,33] := 0.3086827;
   DATA[129,34] := 2.0;
   DATA[129,35] := 250.9453;
   DATA[129,36] := 1.665972;
   DATA[129,37] := 189.6949;
   DATA[129,38] := 0.000128152;
   DATA[129,39] := 1.0;
   DATA[130,0] := 2.427057;
   DATA[130,1] := 526.0655;
   DATA[130,2] := 2.0;
   DATA[130,3] := 2.0;
   DATA[130,4] := 262.1443;
   DATA[130,5] := 8.39163;
   DATA[130,6] := 328.4286;
   DATA[130,7] := 2.440137;
   DATA[130,8] := 2.0;
   DATA[130,9] := 2.0;
   DATA[130,10] := 2.0;
   DATA[130,11] := 19.74198;
   DATA[130,12] := 2.210294;
   DATA[130,13] := 961.1318;
   DATA[130,14] := 1.0;
   DATA[130,15] := 2.0;
   DATA[130,16] := 1.0;
   DATA[130,17] := 1.0;
   DATA[130,18] := 1.0;
   DATA[130,19] := 2.0;
   DATA[130,20] := 148.808;
   DATA[130,21] := 155.7806;
   DATA[130,22] := 1.715824;
   DATA[130,23] := 955.8703;
   DATA[130,24] := 2.0;
   DATA[130,25] := 2.0;
   DATA[130,26] := 7.877019;
   DATA[130,27] := 145.1423;
   DATA[130,28] := 264.2912;
   DATA[130,29] := 12.07383;
   DATA[130,30] := 1.727506;
   DATA[130,31] := 1.280902;
   DATA[130,32] := 0.7353967;
   DATA[130,33] := 0.3086827;
   DATA[130,34] := 2.0;
   DATA[130,35] := 250.9453;
   DATA[130,36] := 1.665972;
   DATA[130,37] := 189.6949;
   DATA[130,38] := 0.000128152;
   DATA[130,39] := 1.0;
   DATA[131,0] := 2.424174;
   DATA[131,1] := 526.8898;
   DATA[131,2] := 2.0;
   DATA[131,3] := 2.0;
   DATA[131,4] := 262.1443;
   DATA[131,5] := 8.39163;
   DATA[131,6] := 328.4286;
   DATA[131,7] := 2.443085;
   DATA[131,8] := 2.0;
   DATA[131,9] := 2.0;
   DATA[131,10] := 2.0;
   DATA[131,11] := 19.74198;
   DATA[131,12] := 2.210294;
   DATA[131,13] := 961.332;
   DATA[131,14] := 1.0;
   DATA[131,15] := 2.0;
   DATA[131,16] := 1.0;
   DATA[131,17] := 1.0;
   DATA[131,18] := 1.0;
   DATA[131,19] := 2.0;
   DATA[131,20] := 148.808;
   DATA[131,21] := 155.7806;
   DATA[131,22] := 1.716592;
   DATA[131,23] := 956.3317;
   DATA[131,24] := 2.0;
   DATA[131,25] := 2.0;
   DATA[131,26] := 7.877019;
   DATA[131,27] := 145.1423;
   DATA[131,28] := 264.2592;
   DATA[131,29] := 12.07383;
   DATA[131,30] := 1.728275;
   DATA[131,31] := 1.281798;
   DATA[131,32] := 0.7353967;
   DATA[131,33] := 0.3069532;
   DATA[131,34] := 2.0;
   DATA[131,35] := 250.9453;
   DATA[131,36] := 1.665972;
   DATA[131,37] := 189.6949;
   DATA[131,38] := 0.000128152;
   DATA[131,39] := 1.0;
   DATA[132,0] := 2.452359;
   DATA[132,1] := 527.1646;
   DATA[132,2] := 2.0;
   DATA[132,3] := 2.0;
   DATA[132,4] := 262.1443;
   DATA[132,5] := 8.39163;
   DATA[132,6] := 328.4286;
   DATA[132,7] := 2.443597;
   DATA[132,8] := 2.0;
   DATA[132,9] := 2.0;
   DATA[132,10] := 2.0;
   DATA[132,11] := 19.70677;
   DATA[132,12] := 2.212343;
   DATA[132,13] := 961.5724;
   DATA[132,14] := 1.0;
   DATA[132,15] := 2.0;
   DATA[132,16] := 1.0;
   DATA[132,17] := 1.0;
   DATA[132,18] := 1.0;
   DATA[132,19] := 2.0;
   DATA[132,20] := 148.808;
   DATA[132,21] := 155.7806;
   DATA[132,22] := 1.716592;
   DATA[132,23] := 956.2933;
   DATA[132,24] := 2.0;
   DATA[132,25] := 2.0;
   DATA[132,26] := 7.877019;
   DATA[132,27] := 145.1423;
   DATA[132,28] := 264.0989;
   DATA[132,29] := 12.07383;
   DATA[132,30] := 1.728275;
   DATA[132,31] := 1.281798;
   DATA[132,32] := 0.7353967;
   DATA[132,33] := 0.3065689;
   DATA[132,34] := 2.0;
   DATA[132,35] := 250.9773;
   DATA[132,36] := 1.665972;
   DATA[132,37] := 189.6949;
   DATA[132,38] := 0.000128152;
   DATA[132,39] := 1.0;
   DATA[133,0] := 2.501041;
   DATA[133,1] := 527.6748;
   DATA[133,2] := 2.0;
   DATA[133,3] := 2.0;
   DATA[133,4] := 262.1443;
   DATA[133,5] := 8.39163;
   DATA[133,6] := 328.4286;
   DATA[133,7] := 2.443597;
   DATA[133,8] := 2.0;
   DATA[133,9] := 2.0;
   DATA[133,10] := 2.0;
   DATA[133,11] := 19.62994;
   DATA[133,12] := 2.213368;
   DATA[133,13] := 961.8127;
   DATA[133,14] := 1.0;
   DATA[133,15] := 2.0;
   DATA[133,16] := 1.0;
   DATA[133,17] := 1.0;
   DATA[133,18] := 1.0;
   DATA[133,19] := 2.0;
   DATA[133,20] := 148.808;
   DATA[133,21] := 155.7806;
   DATA[133,22] := 1.71813;
   DATA[133,23] := 956.3317;
   DATA[133,24] := 2.0;
   DATA[133,25] := 2.0;
   DATA[133,26] := 7.877019;
   DATA[133,27] := 145.1423;
   DATA[133,28] := 264.0989;
   DATA[133,29] := 12.07383;
   DATA[133,30] := 1.72725;
   DATA[133,31] := 1.281798;
   DATA[133,32] := 0.7353967;
   DATA[133,33] := 0.3065689;
   DATA[133,34] := 2.0;
   DATA[133,35] := 251.0734;
   DATA[133,36] := 1.665972;
   DATA[133,37] := 189.6949;
   DATA[133,38] := 0.000128152;
   DATA[133,39] := 1.0;
   DATA[134,0] := 2.550043;
   DATA[134,1] := 527.5571;
   DATA[134,2] := 2.0;
   DATA[134,3] := 2.0;
   DATA[134,4] := 262.1443;
   DATA[134,5] := 8.39163;
   DATA[134,6] := 328.4286;
   DATA[134,7] := 2.443597;
   DATA[134,8] := 2.0;
   DATA[134,9] := 2.0;
   DATA[134,10] := 2.0;
   DATA[134,11] := 19.60433;
   DATA[134,12] := 2.213368;
   DATA[134,13] := 961.8127;
   DATA[134,14] := 1.0;
   DATA[134,15] := 2.0;
   DATA[134,16] := 1.0;
   DATA[134,17] := 1.0;
   DATA[134,18] := 1.0;
   DATA[134,19] := 2.0;
   DATA[134,20] := 148.808;
   DATA[134,21] := 155.7806;
   DATA[134,22] := 1.719027;
   DATA[134,23] := 956.4471;
   DATA[134,24] := 2.0;
   DATA[134,25] := 2.0;
   DATA[134,26] := 7.877019;
   DATA[134,27] := 145.1423;
   DATA[134,28] := 264.0989;
   DATA[134,29] := 12.07383;
   DATA[134,30] := 1.72725;
   DATA[134,31] := 1.281798;
   DATA[134,32] := 0.7380853;
   DATA[134,33] := 0.3084905;
   DATA[134,34] := 2.0;
   DATA[134,35] := 251.0734;
   DATA[134,36] := 1.665972;
   DATA[134,37] := 189.759;
   DATA[134,38] := 0.000128152;
   DATA[134,39] := 1.0;
   DATA[135,0] := 2.576306;
   DATA[135,1] := 527.4001;
   DATA[135,2] := 2.0;
   DATA[135,3] := 2.0;
   DATA[135,4] := 262.1443;
   DATA[135,5] := 8.39163;
   DATA[135,6] := 328.4286;
   DATA[135,7] := 2.4427;
   DATA[135,8] := 2.0;
   DATA[135,9] := 2.0;
   DATA[135,10] := 2.0;
   DATA[135,11] := 19.58832;
   DATA[135,12] := 2.210678;
   DATA[135,13] := 962.4536;
   DATA[135,14] := 1.0;
   DATA[135,15] := 2.0;
   DATA[135,16] := 1.0;
   DATA[135,17] := 1.0;
   DATA[135,18] := 1.0;
   DATA[135,19] := 2.0;
   DATA[135,20] := 148.808;
   DATA[135,21] := 155.7806;
   DATA[135,22] := 1.717233;
   DATA[135,23] := 956.4086;
   DATA[135,24] := 2.0;
   DATA[135,25] := 2.0;
   DATA[135,26] := 7.877019;
   DATA[135,27] := 145.1423;
   DATA[135,28] := 264.0989;
   DATA[135,29] := 12.07383;
   DATA[135,30] := 1.72725;
   DATA[135,31] := 1.290893;
   DATA[135,32] := 0.7380853;
   DATA[135,33] := 0.3084905;
   DATA[135,34] := 2.0;
   DATA[135,35] := 251.0734;
   DATA[135,36] := 1.665972;
   DATA[135,37] := 189.759;
   DATA[135,38] := 0.000128152;
   DATA[135,39] := 1.0;
   DATA[136,0] := 2.619223;
   DATA[136,1] := 526.8505;
   DATA[136,2] := 2.0;
   DATA[136,3] := 2.0;
   DATA[136,4] := 262.1443;
   DATA[136,5] := 8.39163;
   DATA[136,6] := 328.4286;
   DATA[136,7] := 2.439881;
   DATA[136,8] := 2.0;
   DATA[136,9] := 2.0;
   DATA[136,10] := 2.0;
   DATA[136,11] := 19.58832;
   DATA[136,12] := 2.210678;
   DATA[136,13] := 962.5337;
   DATA[136,14] := 1.0;
   DATA[136,15] := 2.0;
   DATA[136,16] := 1.0;
   DATA[136,17] := 1.0;
   DATA[136,18] := 1.0;
   DATA[136,19] := 2.0;
   DATA[136,20] := 148.808;
   DATA[136,21] := 155.7806;
   DATA[136,22] := 1.716208;
   DATA[136,23] := 956.0626;
   DATA[136,24] := 2.0;
   DATA[136,25] := 2.0;
   DATA[136,26] := 7.875737;
   DATA[136,27] := 145.1423;
   DATA[136,28] := 264.131;
   DATA[136,29] := 12.07383;
   DATA[136,30] := 1.72725;
   DATA[136,31] := 1.291277;
   DATA[136,32] := 0.7366771;
   DATA[136,33] := 0.3084905;
   DATA[136,34] := 2.0;
   DATA[136,35] := 251.0734;
   DATA[136,36] := 1.665972;
   DATA[136,37] := 189.7751;
   DATA[136,38] := 0.000128152;
   DATA[136,39] := 1.0;
   DATA[137,0] := 2.644525;
   DATA[137,1] := 526.8505;
   DATA[137,2] := 2.0;
   DATA[137,3] := 2.0;
   DATA[137,4] := 262.1443;
   DATA[137,5] := 8.39163;
   DATA[137,6] := 328.4286;
   DATA[137,7] := 2.439881;
   DATA[137,8] := 2.0;
   DATA[137,9] := 2.0;
   DATA[137,10] := 2.0;
   DATA[137,11] := 19.58832;
   DATA[137,12] := 2.21324;
   DATA[137,13] := 962.7339;
   DATA[137,14] := 1.0;
   DATA[137,15] := 2.0;
   DATA[137,16] := 1.0;
   DATA[137,17] := 1.0;
   DATA[137,18] := 1.0;
   DATA[137,19] := 2.0;
   DATA[137,20] := 148.808;
   DATA[137,21] := 155.7806;
   DATA[137,22] := 1.716208;
   DATA[137,23] := 955.8703;
   DATA[137,24] := 2.0;
   DATA[137,25] := 2.0;
   DATA[137,26] := 7.874455;
   DATA[137,27] := 145.1423;
   DATA[137,28] := 264.163;
   DATA[137,29] := 12.07383;
   DATA[137,30] := 1.728275;
   DATA[137,31] := 1.282183;
   DATA[137,32] := 0.736421;
   DATA[137,33] := 0.3084905;
   DATA[137,34] := 2.0;
   DATA[137,35] := 251.0734;
   DATA[137,36] := 1.665972;
   DATA[137,37] := 189.7751;
   DATA[137,38] := 0.000128152;
   DATA[137,39] := 1.0;
   DATA[138,0] := 2.668225;
   DATA[138,1] := 526.2617;
   DATA[138,2] := 2.0;
   DATA[138,3] := 2.0;
   DATA[138,4] := 262.1443;
   DATA[138,5] := 8.39163;
   DATA[138,6] := 328.4286;
   DATA[138,7] := 2.439881;
   DATA[138,8] := 2.0;
   DATA[138,9] := 2.0;
   DATA[138,10] := 2.0;
   DATA[138,11] := 19.66195;
   DATA[138,12] := 2.212343;
   DATA[138,13] := 962.774;
   DATA[138,14] := 1.0;
   DATA[138,15] := 2.0;
   DATA[138,16] := 1.0;
   DATA[138,17] := 1.0;
   DATA[138,18] := 1.0;
   DATA[138,19] := 2.0;
   DATA[138,20] := 148.808;
   DATA[138,21] := 155.7806;
   DATA[138,22] := 1.716208;
   DATA[138,23] := 955.3704;
   DATA[138,24] := 2.0;
   DATA[138,25] := 2.0;
   DATA[138,26] := 7.874455;
   DATA[138,27] := 145.1423;
   DATA[138,28] := 264.2271;
   DATA[138,29] := 12.07383;
   DATA[138,30] := 1.728275;
   DATA[138,31] := 1.269502;
   DATA[138,32] := 0.736421;
   DATA[138,33] := 0.3084905;
   DATA[138,34] := 2.0;
   DATA[138,35] := 251.0734;
   DATA[138,36] := 1.665972;
   DATA[138,37] := 189.7751;
   DATA[138,38] := 0.000128152;
   DATA[138,39] := 1.0;
   DATA[139,0] := 2.668225;
   DATA[139,1] := 526.2617;
   DATA[139,2] := 2.0;
   DATA[139,3] := 2.0;
   DATA[139,4] := 262.1443;
   DATA[139,5] := 8.39163;
   DATA[139,6] := 328.4286;
   DATA[139,7] := 2.439881;
   DATA[139,8] := 2.0;
   DATA[139,9] := 2.0;
   DATA[139,10] := 2.0;
   DATA[139,11] := 19.66195;
   DATA[139,12] := 2.212343;
   DATA[139,13] := 962.774;
   DATA[139,14] := 1.0;
   DATA[139,15] := 2.0;
   DATA[139,16] := 1.0;
   DATA[139,17] := 1.0;
   DATA[139,18] := 1.0;
   DATA[139,19] := 2.0;
   DATA[139,20] := 148.808;
   DATA[139,21] := 155.7806;
   DATA[139,22] := 1.716208;
   DATA[139,23] := 955.3704;
   DATA[139,24] := 2.0;
   DATA[139,25] := 2.0;
   DATA[139,26] := 7.874455;
   DATA[139,27] := 145.1423;
   DATA[139,28] := 264.2271;
   DATA[139,29] := 12.07383;
   DATA[139,30] := 1.728275;
   DATA[139,31] := 1.269502;
   DATA[139,32] := 0.736421;
   DATA[139,33] := 0.3084905;
   DATA[139,34] := 2.0;
   DATA[139,35] := 251.0734;
   DATA[139,36] := 1.665972;
   DATA[139,37] := 189.7751;
   DATA[139,38] := 0.000128152;
   DATA[139,39] := 1.0;
   DATA[140,0] := 2.671748;
   DATA[140,1] := 525.5944;
   DATA[140,2] := 2.0;
   DATA[140,3] := 2.0;
   DATA[140,4] := 262.1443;
   DATA[140,5] := 8.39163;
   DATA[140,6] := 328.2748;
   DATA[140,7] := 2.439881;
   DATA[140,8] := 2.0;
   DATA[140,9] := 2.0;
   DATA[140,10] := 2.0;
   DATA[140,11] := 19.66195;
   DATA[140,12] := 2.21055;
   DATA[140,13] := 962.6538;
   DATA[140,14] := 1.0;
   DATA[140,15] := 2.0;
   DATA[140,16] := 1.0;
   DATA[140,17] := 1.0;
   DATA[140,18] := 1.0;
   DATA[140,19] := 2.0;
   DATA[140,20] := 148.808;
   DATA[140,21] := 155.7806;
   DATA[140,22] := 1.716849;
   DATA[140,23] := 955.332;
   DATA[140,24] := 2.0;
   DATA[140,25] := 2.0;
   DATA[140,26] := 7.874455;
   DATA[140,27] := 145.1423;
   DATA[140,28] := 264.2271;
   DATA[140,29] := 12.07383;
   DATA[140,30] := 1.726865;
   DATA[140,31] := 1.261816;
   DATA[140,32] := 0.7348846;
   DATA[140,33] := 0.3084905;
   DATA[140,34] := 2.0;
   DATA[140,35] := 251.0734;
   DATA[140,36] := 1.665972;
   DATA[140,37] := 189.7751;
   DATA[140,38] := 0.000128152;
   DATA[140,39] := 1.0;
   DATA[141,0] := 2.652852;
   DATA[141,1] := 525.3982;
   DATA[141,2] := 2.0;
   DATA[141,3] := 2.0;
   DATA[141,4] := 262.1443;
   DATA[141,5] := 8.39163;
   DATA[141,6] := 328.2235;
   DATA[141,7] := 2.439881;
   DATA[141,8] := 2.0;
   DATA[141,9] := 2.0;
   DATA[141,10] := 2.0;
   DATA[141,11] := 19.70037;
   DATA[141,12] := 2.209525;
   DATA[141,13] := 963.2146;
   DATA[141,14] := 1.0;
   DATA[141,15] := 2.0;
   DATA[141,16] := 1.0;
   DATA[141,17] := 1.0;
   DATA[141,18] := 1.0;
   DATA[141,19] := 2.0;
   DATA[141,20] := 148.808;
   DATA[141,21] := 155.9087;
   DATA[141,22] := 1.717233;
   DATA[141,23] := 955.4473;
   DATA[141,24] := 2.0;
   DATA[141,25] := 2.0;
   DATA[141,26] := 7.874455;
   DATA[141,27] := 145.1423;
   DATA[141,28] := 264.2271;
   DATA[141,29] := 12.07383;
   DATA[141,30] := 1.726609;
   DATA[141,31] := 1.270142;
   DATA[141,32] := 0.7348846;
   DATA[141,33] := 0.3084905;
   DATA[141,34] := 2.0;
   DATA[141,35] := 251.0574;
   DATA[141,36] := 1.665972;
   DATA[141,37] := 189.7751;
   DATA[141,38] := 0.000128152;
   DATA[141,39] := 1.0;
   DATA[142,0] := 2.632034;
   DATA[142,1] := 524.8879;
   DATA[142,2] := 2.0;
   DATA[142,3] := 2.0;
   DATA[142,4] := 262.1443;
   DATA[142,5] := 8.39163;
   DATA[142,6] := 328.2235;
   DATA[142,7] := 2.439881;
   DATA[142,8] := 2.0;
   DATA[142,9] := 2.0;
   DATA[142,10] := 2.0;
   DATA[142,11] := 19.70037;
   DATA[142,12] := 2.209525;
   DATA[142,13] := 963.8555;
   DATA[142,14] := 1.0;
   DATA[142,15] := 2.0;
   DATA[142,16] := 1.0;
   DATA[142,17] := 1.0;
   DATA[142,18] := 1.0;
   DATA[142,19] := 2.0;
   DATA[142,20] := 148.808;
   DATA[142,21] := 155.9087;
   DATA[142,22] := 1.717233;
   DATA[142,23] := 955.4473;
   DATA[142,24] := 2.0;
   DATA[142,25] := 2.0;
   DATA[142,26] := 7.874455;
   DATA[142,27] := 145.1423;
   DATA[142,28] := 264.2271;
   DATA[142,29] := 12.07383;
   DATA[142,30] := 1.726609;
   DATA[142,31] := 1.28705;
   DATA[142,32] := 0.7348846;
   DATA[142,33] := 0.3077219;
   DATA[142,34] := 2.0;
   DATA[142,35] := 250.9453;
   DATA[142,36] := 1.665972;
   DATA[142,37] := 189.5828;
   DATA[142,38] := 0.000128152;
   DATA[142,39] := 1.0;
   DATA[143,0] := 2.628831;
   DATA[143,1] := 524.7309;
   DATA[143,2] := 2.0;
   DATA[143,3] := 2.0;
   DATA[143,4] := 262.0802;
   DATA[143,5] := 8.39163;
   DATA[143,6] := 328.2235;
   DATA[143,7] := 2.439881;
   DATA[143,8] := 2.0;
   DATA[143,9] := 2.0;
   DATA[143,10] := 2.0;
   DATA[143,11] := 19.70037;
   DATA[143,12] := 2.209525;
   DATA[143,13] := 964.0557;
   DATA[143,14] := 1.0;
   DATA[143,15] := 2.0;
   DATA[143,16] := 1.0;
   DATA[143,17] := 1.0;
   DATA[143,18] := 1.0;
   DATA[143,19] := 2.0;
   DATA[143,20] := 148.808;
   DATA[143,21] := 155.9087;
   DATA[143,22] := 1.717233;
   DATA[143,23] := 955.4473;
   DATA[143,24] := 2.0;
   DATA[143,25] := 2.0;
   DATA[143,26] := 7.87766;
   DATA[143,27] := 145.1423;
   DATA[143,28] := 264.2271;
   DATA[143,29] := 12.07383;
   DATA[143,30] := 1.726609;
   DATA[143,31] := 1.285385;
   DATA[143,32] := 0.7348846;
   DATA[143,33] := 0.3072094;
   DATA[143,34] := 2.0;
   DATA[143,35] := 250.9453;
   DATA[143,36] := 1.665972;
   DATA[143,37] := 189.5828;
   DATA[143,38] := 0.000128152;
   DATA[143,39] := 1.0;
   DATA[144,0] := 2.628511;
   DATA[144,1] := 524.8879;
   DATA[144,2] := 2.0;
   DATA[144,3] := 2.0;
   DATA[144,4] := 262.0802;
   DATA[144,5] := 8.39163;
   DATA[144,6] := 328.3004;
   DATA[144,7] := 2.439881;
   DATA[144,8] := 2.0;
   DATA[144,9] := 2.0;
   DATA[144,10] := 2.0;
   DATA[144,11] := 19.71637;
   DATA[144,12] := 2.209525;
   DATA[144,13] := 963.9355;
   DATA[144,14] := 1.0;
   DATA[144,15] := 2.0;
   DATA[144,16] := 1.0;
   DATA[144,17] := 1.0;
   DATA[144,18] := 1.0;
   DATA[144,19] := 2.0;
   DATA[144,20] := 148.808;
   DATA[144,21] := 155.9087;
   DATA[144,22] := 1.717233;
   DATA[144,23] := 955.332;
   DATA[144,24] := 2.0;
   DATA[144,25] := 2.0;
   DATA[144,26] := 7.87766;
   DATA[144,27] := 145.1423;
   DATA[144,28] := 264.2271;
   DATA[144,29] := 12.07383;
   DATA[144,30] := 1.726609;
   DATA[144,31] := 1.281927;
   DATA[144,32] := 0.7348846;
   DATA[144,33] := 0.3072094;
   DATA[144,34] := 2.0;
   DATA[144,35] := 250.9453;
   DATA[144,36] := 1.665972;
   DATA[144,37] := 189.5828;
   DATA[144,38] := 0.000128152;
   DATA[144,39] := 1.0;
   DATA[145,0] := 2.61602;
   DATA[145,1] := 525.1234;
   DATA[145,2] := 2.0;
   DATA[145,3] := 2.0;
   DATA[145,4] := 262.0802;
   DATA[145,5] := 8.39163;
   DATA[145,6] := 328.4286;
   DATA[145,7] := 2.439881;
   DATA[145,8] := 2.0;
   DATA[145,9] := 2.0;
   DATA[145,10] := 2.0;
   DATA[145,11] := 19.73558;
   DATA[145,12] := 2.209525;
   DATA[145,13] := 963.8555;
   DATA[145,14] := 1.0;
   DATA[145,15] := 2.0;
   DATA[145,16] := 1.0;
   DATA[145,17] := 1.0;
   DATA[145,18] := 1.0;
   DATA[145,19] := 2.0;
   DATA[145,20] := 148.808;
   DATA[145,21] := 155.9087;
   DATA[145,22] := 1.717233;
   DATA[145,23] := 955.2935;
   DATA[145,24] := 2.0;
   DATA[145,25] := 2.0;
   DATA[145,26] := 7.87766;
   DATA[145,27] := 145.1423;
   DATA[145,28] := 264.2271;
   DATA[145,29] := 12.41989;
   DATA[145,30] := 1.726609;
   DATA[145,31] := 1.281927;
   DATA[145,32] := 0.7348846;
   DATA[145,33] := 0.306761;
   DATA[145,34] := 2.0;
   DATA[145,35] := 250.9453;
   DATA[145,36] := 1.665972;
   DATA[145,37] := 189.5828;
   DATA[145,38] := 0.000128152;
   DATA[145,39] := 1.0;
   DATA[146,0] := 2.597124;
   DATA[146,1] := 525.2019;
   DATA[146,2] := 2.0;
   DATA[146,3] := 2.0;
   DATA[146,4] := 262.0802;
   DATA[146,5] := 8.39163;
   DATA[146,6] := 328.5055;
   DATA[146,7] := 2.439881;
   DATA[146,8] := 2.0;
   DATA[146,9] := 2.0;
   DATA[146,10] := 2.0;
   DATA[146,11] := 19.73558;
   DATA[146,12] := 2.209525;
   DATA[146,13] := 963.535;
   DATA[146,14] := 1.0;
   DATA[146,15] := 2.0;
   DATA[146,16] := 1.0;
   DATA[146,17] := 1.0;
   DATA[146,18] := 1.0;
   DATA[146,19] := 2.0;
   DATA[146,20] := 148.808;
   DATA[146,21] := 155.9087;
   DATA[146,22] := 1.717233;
   DATA[146,23] := 955.332;
   DATA[146,24] := 2.0;
   DATA[146,25] := 2.0;
   DATA[146,26] := 7.87766;
   DATA[146,27] := 145.1423;
   DATA[146,28] := 264.2271;
   DATA[146,29] := 12.41989;
   DATA[146,30] := 1.726609;
   DATA[146,31] := 1.281927;
   DATA[146,32] := 0.7348846;
   DATA[146,33] := 0.3065048;
   DATA[146,34] := 2.0;
   DATA[146,35] := 250.9453;
   DATA[146,36] := 1.665972;
   DATA[146,37] := 189.7751;
   DATA[146,38] := 0.000128152;
   DATA[146,39] := 1.0;
   DATA[147,0] := 2.575986;
   DATA[147,1] := 525.2804;
   DATA[147,2] := 2.0;
   DATA[147,3] := 2.0;
   DATA[147,4] := 262.0802;
   DATA[147,5] := 8.39163;
   DATA[147,6] := 328.5055;
   DATA[147,7] := 2.440393;
   DATA[147,8] := 2.0;
   DATA[147,9] := 2.0;
   DATA[147,10] := 2.0;
   DATA[147,11] := 19.73558;
   DATA[147,12] := 2.209525;
   DATA[147,13] := 963.2146;
   DATA[147,14] := 1.0;
   DATA[147,15] := 2.0;
   DATA[147,16] := 1.0;
   DATA[147,17] := 1.0;
   DATA[147,18] := 1.0;
   DATA[147,19] := 2.0;
   DATA[147,20] := 148.808;
   DATA[147,21] := 155.9087;
   DATA[147,22] := 1.717233;
   DATA[147,23] := 955.332;
   DATA[147,24] := 2.0;
   DATA[147,25] := 2.0;
   DATA[147,26] := 7.87766;
   DATA[147,27] := 145.1423;
   DATA[147,28] := 264.2271;
   DATA[147,29] := 12.11228;
   DATA[147,30] := 1.726609;
   DATA[147,31] := 1.296401;
   DATA[147,32] := 0.7348846;
   DATA[147,33] := 0.3089389;
   DATA[147,34] := 2.0;
   DATA[147,35] := 250.9453;
   DATA[147,36] := 1.665972;
   DATA[147,37] := 189.8391;
   DATA[147,38] := 0.000128152;
   DATA[147,39] := 1.0;
   DATA[148,0] := 2.559331;
   DATA[148,1] := 525.3196;
   DATA[148,2] := 2.0;
   DATA[148,3] := 2.0;
   DATA[148,4] := 262.0802;
   DATA[148,5] := 8.39163;
   DATA[148,6] := 328.1723;
   DATA[148,7] := 2.440393;
   DATA[148,8] := 2.0;
   DATA[148,9] := 2.0;
   DATA[148,10] := 2.0;
   DATA[148,11] := 19.73558;
   DATA[148,12] := 2.209525;
   DATA[148,13] := 963.6552;
   DATA[148,14] := 1.0;
   DATA[148,15] := 2.0;
   DATA[148,16] := 1.0;
   DATA[148,17] := 1.0;
   DATA[148,18] := 1.0;
   DATA[148,19] := 2.0;
   DATA[148,20] := 148.808;
   DATA[148,21] := 155.9087;
   DATA[148,22] := 1.717233;
   DATA[148,23] := 955.1782;
   DATA[148,24] := 2.0;
   DATA[148,25] := 2.0;
   DATA[148,26] := 7.87766;
   DATA[148,27] := 145.1423;
   DATA[148,28] := 264.2271;
   DATA[148,29] := 12.03538;
   DATA[148,30] := 1.726609;
   DATA[148,31] := 1.310491;
   DATA[148,32] := 0.7348846;
   DATA[148,33] := 0.3089389;
   DATA[148,34] := 2.0;
   DATA[148,35] := 250.9453;
   DATA[148,36] := 1.665972;
   DATA[148,37] := 189.8391;
   DATA[148,38] := 0.000128152;
   DATA[148,39] := 1.0;
   DATA[149,0] := 2.542677;
   DATA[149,1] := 525.4374;
   DATA[149,2] := 2.0;
   DATA[149,3] := 2.0;
   DATA[149,4] := 262.0802;
   DATA[149,5] := 8.39163;
   DATA[149,6] := 328.121;
   DATA[149,7] := 2.440393;
   DATA[149,8] := 2.0;
   DATA[149,9] := 2.0;
   DATA[149,10] := 2.0;
   DATA[149,11] := 19.73558;
   DATA[149,12] := 2.208756;
   DATA[149,13] := 963.6151;
   DATA[149,14] := 1.0;
   DATA[149,15] := 2.0;
   DATA[149,16] := 1.0;
   DATA[149,17] := 1.0;
   DATA[149,18] := 1.0;
   DATA[149,19] := 2.0;
   DATA[149,20] := 148.808;
   DATA[149,21] := 155.9087;
   DATA[149,22] := 1.717233;
   DATA[149,23] := 955.5242;
   DATA[149,24] := 2.0;
   DATA[149,25] := 2.0;
   DATA[149,26] := 7.87766;
   DATA[149,27] := 145.2704;
   DATA[149,28] := 264.2271;
   DATA[149,29] := 12.03538;
   DATA[149,30] := 1.72789;
   DATA[149,31] := 1.311772;
   DATA[149,32] := 0.7348846;
   DATA[149,33] := 0.3089389;
   DATA[149,34] := 2.0;
   DATA[149,35] := 250.9453;
   DATA[149,36] := 1.665972;
   DATA[149,37] := 189.8391;
   DATA[149,38] := 0.000128152;
   DATA[149,39] := 1.0;
   DATA[150,0] := 2.52314;
   DATA[150,1] := 525.4767;
   DATA[150,2] := 2.0;
   DATA[150,3] := 2.0;
   DATA[150,4] := 262.0802;
   DATA[150,5] := 8.39163;
   DATA[150,6] := 328.121;
   DATA[150,7] := 2.440393;
   DATA[150,8] := 2.0;
   DATA[150,9] := 2.0;
   DATA[150,10] := 2.0;
   DATA[150,11] := 19.73558;
   DATA[150,12] := 2.208116;
   DATA[150,13] := 963.6552;
   DATA[150,14] := 1.0;
   DATA[150,15] := 2.0;
   DATA[150,16] := 1.0;
   DATA[150,17] := 1.0;
   DATA[150,18] := 1.0;
   DATA[150,19] := 2.0;
   DATA[150,20] := 148.808;
   DATA[150,21] := 155.9087;
   DATA[150,22] := 1.717233;
   DATA[150,23] := 955.2551;
   DATA[150,24] := 2.0;
   DATA[150,25] := 2.0;
   DATA[150,26] := 7.87766;
   DATA[150,27] := 145.2704;
   DATA[150,28] := 264.2271;
   DATA[150,29] := 12.03538;
   DATA[150,30] := 1.728019;
   DATA[150,31] := 1.300243;
   DATA[150,32] := 0.7348846;
   DATA[150,33] := 0.3083624;
   DATA[150,34] := 2.0;
   DATA[150,35] := 251.0734;
   DATA[150,36] := 1.665972;
   DATA[150,37] := 189.8391;
   DATA[150,38] := 0.000128152;
   DATA[150,39] := 1.0;
   DATA[151,0] := 2.509048;
   DATA[151,1] := 525.83;
   DATA[151,2] := 2.0;
   DATA[151,3] := 2.0;
   DATA[151,4] := 262.0802;
   DATA[151,5] := 8.39163;
   DATA[151,6] := 328.121;
   DATA[151,7] := 2.440393;
   DATA[151,8] := 2.0;
   DATA[151,9] := 2.0;
   DATA[151,10] := 2.0;
   DATA[151,11] := 19.69396;
   DATA[151,12] := 2.208116;
   DATA[151,13] := 964.1759;
   DATA[151,14] := 1.0;
   DATA[151,15] := 2.0;
   DATA[151,16] := 1.0;
   DATA[151,17] := 1.0;
   DATA[151,18] := 1.0;
   DATA[151,19] := 2.0;
   DATA[151,20] := 148.808;
   DATA[151,21] := 155.9087;
   DATA[151,22] := 1.718643;
   DATA[151,23] := 955.6396;
   DATA[151,24] := 2.0;
   DATA[151,25] := 2.0;
   DATA[151,26] := 7.876058;
   DATA[151,27] := 145.2704;
   DATA[151,28] := 264.2271;
   DATA[151,29] := 12.03538;
   DATA[151,30] := 1.728019;
   DATA[151,31] := 1.292558;
   DATA[151,32] := 0.7348846;
   DATA[151,33] := 0.3083624;
   DATA[151,34] := 2.0;
   DATA[151,35] := 251.1215;
   DATA[151,36] := 1.665972;
   DATA[151,37] := 189.8391;
   DATA[151,38] := 0.000128152;
   DATA[151,39] := 1.0;
   DATA[152,0] := 2.495596;
   DATA[152,1] := 525.7907;
   DATA[152,2] := 2.0;
   DATA[152,3] := 2.0;
   DATA[152,4] := 262.0802;
   DATA[152,5] := 8.39163;
   DATA[152,6] := 328.121;
   DATA[152,7] := 2.440393;
   DATA[152,8] := 2.0;
   DATA[152,9] := 2.0;
   DATA[152,10] := 2.0;
   DATA[152,11] := 19.68756;
   DATA[152,12] := 2.208116;
   DATA[152,13] := 963.9355;
   DATA[152,14] := 1.0;
   DATA[152,15] := 2.0;
   DATA[152,16] := 1.0;
   DATA[152,17] := 1.0;
   DATA[152,18] := 1.0;
   DATA[152,19] := 2.0;
   DATA[152,20] := 148.808;
   DATA[152,21] := 155.9087;
   DATA[152,22] := 1.718643;
   DATA[152,23] := 955.9472;
   DATA[152,24] := 2.0;
   DATA[152,25] := 2.0;
   DATA[152,26] := 7.874135;
   DATA[152,27] := 145.2704;
   DATA[152,28] := 264.2271;
   DATA[152,29] := 12.03538;
   DATA[152,30] := 1.728019;
   DATA[152,31] := 1.291405;
   DATA[152,32] := 0.7348846;
   DATA[152,33] := 0.3083624;
   DATA[152,34] := 2.0;
   DATA[152,35] := 251.1215;
   DATA[152,36] := 1.665972;
   DATA[152,37] := 189.8391;
   DATA[152,38] := 0.000128152;
   DATA[152,39] := 1.0;
   DATA[153,0] := 2.483426;
   DATA[153,1] := 525.83;
   DATA[153,2] := 2.0;
   DATA[153,3] := 2.0;
   DATA[153,4] := 262.0802;
   DATA[153,5] := 8.39163;
   DATA[153,6] := 328.121;
   DATA[153,7] := 2.440393;
   DATA[153,8] := 2.0;
   DATA[153,9] := 2.0;
   DATA[153,10] := 2.0;
   DATA[153,11] := 19.68756;
   DATA[153,12] := 2.208884;
   DATA[153,13] := 963.7353;
   DATA[153,14] := 1.0;
   DATA[153,15] := 2.0;
   DATA[153,16] := 1.0;
   DATA[153,17] := 1.0;
   DATA[153,18] := 1.0;
   DATA[153,19] := 2.0;
   DATA[153,20] := 148.808;
   DATA[153,21] := 155.9087;
   DATA[153,22] := 1.718643;
   DATA[153,23] := 956.0626;
   DATA[153,24] := 2.0;
   DATA[153,25] := 2.0;
   DATA[153,26] := 7.874135;
   DATA[153,27] := 145.2704;
   DATA[153,28] := 264.2271;
   DATA[153,29] := 12.03538;
   DATA[153,30] := 1.726865;
   DATA[153,31] := 1.291405;
   DATA[153,32] := 0.7348846;
   DATA[153,33] := 0.3083624;
   DATA[153,34] := 2.0;
   DATA[153,35] := 251.0414;
   DATA[153,36] := 1.665972;
   DATA[153,37] := 189.6789;
   DATA[153,38] := 0.000128152;
   DATA[153,39] := 1.0;
   DATA[154,0] := 2.46549;
   DATA[154,1] := 525.8692;
   DATA[154,2] := 2.0;
   DATA[154,3] := 2.0;
   DATA[154,4] := 262.0802;
   DATA[154,5] := 8.39163;
   DATA[154,6] := 328.121;
   DATA[154,7] := 2.440393;
   DATA[154,8] := 2.0;
   DATA[154,9] := 2.0;
   DATA[154,10] := 2.0;
   DATA[154,11] := 19.74198;
   DATA[154,12] := 2.209653;
   DATA[154,13] := 964.256;
   DATA[154,14] := 1.0;
   DATA[154,15] := 2.0;
   DATA[154,16] := 1.0;
   DATA[154,17] := 1.0;
   DATA[154,18] := 1.0;
   DATA[154,19] := 2.0;
   DATA[154,20] := 148.808;
   DATA[154,21] := 155.9087;
   DATA[154,22] := 1.716849;
   DATA[154,23] := 956.0241;
   DATA[154,24] := 2.0;
   DATA[154,25] := 2.0;
   DATA[154,26] := 7.874135;
   DATA[154,27] := 145.2704;
   DATA[154,28] := 264.2271;
   DATA[154,29] := 12.03538;
   DATA[154,30] := 1.726865;
   DATA[154,31] := 1.300884;
   DATA[154,32] := 0.7351407;
   DATA[154,33] := 0.3083624;
   DATA[154,34] := 2.0;
   DATA[154,35] := 250.8331;
   DATA[154,36] := 1.665972;
   DATA[154,37] := 189.6789;
   DATA[154,38] := 0.000128152;
   DATA[154,39] := 1.0;
   DATA[155,0] := 2.450758;
   DATA[155,1] := 525.9869;
   DATA[155,2] := 2.0;
   DATA[155,3] := 2.0;
   DATA[155,4] := 262.0802;
   DATA[155,5] := 8.39163;
   DATA[155,6] := 328.1466;
   DATA[155,7] := 2.440393;
   DATA[155,8] := 2.0;
   DATA[155,9] := 2.0;
   DATA[155,10] := 2.0;
   DATA[155,11] := 19.74198;
   DATA[155,12] := 2.209653;
   DATA[155,13] := 964.3762;
   DATA[155,14] := 1.0;
   DATA[155,15] := 2.0;
   DATA[155,16] := 1.0;
   DATA[155,17] := 1.0;
   DATA[155,18] := 1.0;
   DATA[155,19] := 2.0;
   DATA[155,20] := 148.808;
   DATA[155,21] := 155.9087;
   DATA[155,22] := 1.716464;
   DATA[155,23] := 955.7549;
   DATA[155,24] := 2.0;
   DATA[155,25] := 2.0;
   DATA[155,26] := 7.874135;
   DATA[155,27] := 145.2704;
   DATA[155,28] := 264.2271;
   DATA[155,29] := 12.03538;
   DATA[155,30] := 1.724942;
   DATA[155,31] := 1.29307;
   DATA[155,32] := 0.7359089;
   DATA[155,33] := 0.3083624;
   DATA[155,34] := 2.0;
   DATA[155,35] := 250.8331;
   DATA[155,36] := 1.665972;
   DATA[155,37] := 189.6789;
   DATA[155,38] := 0.000128152;
   DATA[155,39] := 1.0;
   DATA[156,0] := 2.429619;
   DATA[156,1] := 525.9084;
   DATA[156,2] := 2.0;
   DATA[156,3] := 2.0;
   DATA[156,4] := 262.0802;
   DATA[156,5] := 8.39163;
   DATA[156,6] := 328.2748;
   DATA[156,7] := 2.441547;
   DATA[156,8] := 2.0;
   DATA[156,9] := 2.0;
   DATA[156,10] := 2.0;
   DATA[156,11] := 19.74198;
   DATA[156,12] := 2.2126;
   DATA[156,13] := 964.5764;
   DATA[156,14] := 1.0;
   DATA[156,15] := 2.0;
   DATA[156,16] := 1.0;
   DATA[156,17] := 1.0;
   DATA[156,18] := 1.0;
   DATA[156,19] := 2.0;
   DATA[156,20] := 148.808;
   DATA[156,21] := 155.9087;
   DATA[156,22] := 1.71608;
   DATA[156,23] := 955.7165;
   DATA[156,24] := 2.0;
   DATA[156,25] := 2.0;
   DATA[156,26] := 7.876378;
   DATA[156,27] := 145.2704;
   DATA[156,28] := 264.2271;
   DATA[156,29] := 12.03538;
   DATA[156,30] := 1.724942;
   DATA[156,31] := 1.291789;
   DATA[156,32] := 0.7359089;
   DATA[156,33] := 0.3083624;
   DATA[156,34] := 2.0;
   DATA[156,35] := 250.8331;
   DATA[156,36] := 1.665972;
   DATA[156,37] := 189.6789;
   DATA[156,38] := 0.000128152;
   DATA[156,39] := 1.0;
   DATA[157,0] := 2.421932;
   DATA[157,1] := 526.1047;
   DATA[157,2] := 2.0;
   DATA[157,3] := 2.0;
   DATA[157,4] := 262.0802;
   DATA[157,5] := 8.39163;
   DATA[157,6] := 328.2748;
   DATA[157,7] := 2.441803;
   DATA[157,8] := 2.0;
   DATA[157,9] := 2.0;
   DATA[157,10] := 2.0;
   DATA[157,11] := 19.74198;
   DATA[157,12] := 2.212728;
   DATA[157,13] := 964.256;
   DATA[157,14] := 1.0;
   DATA[157,15] := 2.0;
   DATA[157,16] := 1.0;
   DATA[157,17] := 1.0;
   DATA[157,18] := 1.0;
   DATA[157,19] := 2.0;
   DATA[157,20] := 148.808;
   DATA[157,21] := 155.9087;
   DATA[157,22] := 1.71608;
   DATA[157,23] := 955.6396;
   DATA[157,24] := 2.0;
   DATA[157,25] := 2.0;
   DATA[157,26] := 7.876378;
   DATA[157,27] := 145.2704;
   DATA[157,28] := 264.2271;
   DATA[157,29] := 12.26609;
   DATA[157,30] := 1.724942;
   DATA[157,31] := 1.286025;
   DATA[157,32] := 0.7359089;
   DATA[157,33] := 0.3083624;
   DATA[157,34] := 2.0;
   DATA[157,35] := 250.8331;
   DATA[157,36] := 1.665972;
   DATA[157,37] := 189.6789;
   DATA[157,38] := 0.000128152;
   DATA[157,39] := 1.0;
   DATA[158,0] := 2.420651;
   DATA[158,1] := 526.2617;
   DATA[158,2] := 2.0;
   DATA[158,3] := 2.0;
   DATA[158,4] := 262.0802;
   DATA[158,5] := 8.39163;
   DATA[158,6] := 328.2748;
   DATA[158,7] := 2.440521;
   DATA[158,8] := 2.0;
   DATA[158,9] := 2.0;
   DATA[158,10] := 2.0;
   DATA[158,11] := 19.74198;
   DATA[158,12] := 2.21324;
   DATA[158,13] := 963.8555;
   DATA[158,14] := 1.0;
   DATA[158,15] := 2.0;
   DATA[158,16] := 1.0;
   DATA[158,17] := 1.0;
   DATA[158,18] := 1.0;
   DATA[158,19] := 2.0;
   DATA[158,20] := 148.808;
   DATA[158,21] := 155.9087;
   DATA[158,22] := 1.71608;
   DATA[158,23] := 955.5627;
   DATA[158,24] := 2.0;
   DATA[158,25] := 2.0;
   DATA[158,26] := 7.87766;
   DATA[158,27] := 145.2704;
   DATA[158,28] := 264.2271;
   DATA[158,29] := 12.26609;
   DATA[158,30] := 1.724942;
   DATA[158,31] := 1.272704;
   DATA[158,32] := 0.7359089;
   DATA[158,33] := 0.3083624;
   DATA[158,34] := 2.0;
   DATA[158,35] := 250.8331;
   DATA[158,36] := 1.665972;
   DATA[158,37] := 189.6789;
   DATA[158,38] := 0.000128152;
   DATA[158,39] := 1.0;
   DATA[159,0] := 2.420651;
   DATA[159,1] := 526.4188;
   DATA[159,2] := 2.0;
   DATA[159,3] := 2.0;
   DATA[159,4] := 262.0802;
   DATA[159,5] := 8.39163;
   DATA[159,6] := 328.2748;
   DATA[159,7] := 2.440137;
   DATA[159,8] := 2.0;
   DATA[159,9] := 2.0;
   DATA[159,10] := 2.0;
   DATA[159,11] := 19.74198;
   DATA[159,12] := 2.21324;
   DATA[159,13] := 963.8154;
   DATA[159,14] := 1.0;
   DATA[159,15] := 2.0;
   DATA[159,16] := 1.0;
   DATA[159,17] := 1.0;
   DATA[159,18] := 1.0;
   DATA[159,19] := 2.0;
   DATA[159,20] := 148.808;
   DATA[159,21] := 155.9087;
   DATA[159,22] := 1.71608;
   DATA[159,23] := 955.3704;
   DATA[159,24] := 2.0;
   DATA[159,25] := 2.0;
   DATA[159,26] := 7.87766;
   DATA[159,27] := 145.2704;
   DATA[159,28] := 264.2271;
   DATA[159,29] := 12.26609;
   DATA[159,30] := 1.724942;
   DATA[159,31] := 1.271295;
   DATA[159,32] := 0.7359089;
   DATA[159,33] := 0.3083624;
   DATA[159,34] := 2.0;
   DATA[159,35] := 250.8331;
   DATA[159,36] := 1.665972;
   DATA[159,37] := 189.6789;
   DATA[159,38] := 0.000128152;
   DATA[159,39] := 1.0;
   DATA[160,0] := 2.463248;
   DATA[160,1] := 526.301;
   DATA[160,2] := 2.0;
   DATA[160,3] := 2.0;
   DATA[160,4] := 262.0802;
   DATA[160,5] := 8.39163;
   DATA[160,6] := 328.2748;
   DATA[160,7] := 2.440137;
   DATA[160,8] := 2.0;
   DATA[160,9] := 2.0;
   DATA[160,10] := 2.0;
   DATA[160,11] := 19.74198;
   DATA[160,12] := 2.21324;
   DATA[160,13] := 963.3748;
   DATA[160,14] := 1.0;
   DATA[160,15] := 2.0;
   DATA[160,16] := 1.0;
   DATA[160,17] := 1.0;
   DATA[160,18] := 1.0;
   DATA[160,19] := 2.0;
   DATA[160,20] := 148.808;
   DATA[160,21] := 155.9087;
   DATA[160,22] := 1.71608;
   DATA[160,23] := 955.3704;
   DATA[160,24] := 2.0;
   DATA[160,25] := 2.0;
   DATA[160,26] := 7.87766;
   DATA[160,27] := 145.1423;
   DATA[160,28] := 264.2271;
   DATA[160,29] := 12.26609;
   DATA[160,30] := 1.726737;
   DATA[160,31] := 1.271295;
   DATA[160,32] := 0.7351407;
   DATA[160,33] := 0.3082983;
   DATA[160,34] := 2.0;
   DATA[160,35] := 250.8331;
   DATA[160,36] := 1.649953;
   DATA[160,37] := 189.6789;
   DATA[160,38] := 0.000128152;
   DATA[160,39] := 1.0;
   DATA[161,0] := 2.510009;
   DATA[161,1] := 526.1047;
   DATA[161,2] := 2.0;
   DATA[161,3] := 2.0;
   DATA[161,4] := 262.0802;
   DATA[161,5] := 8.39163;
   DATA[161,6] := 328.2748;
   DATA[161,7] := 2.440137;
   DATA[161,8] := 2.0;
   DATA[161,9] := 2.0;
   DATA[161,10] := 2.0;
   DATA[161,11] := 19.89884;
   DATA[161,12] := 2.21324;
   DATA[161,13] := 963.2546;
   DATA[161,14] := 1.0;
   DATA[161,15] := 2.0;
   DATA[161,16] := 1.0;
   DATA[161,17] := 1.0;
   DATA[161,18] := 1.0;
   DATA[161,19] := 2.0;
   DATA[161,20] := 148.808;
   DATA[161,21] := 155.9087;
   DATA[161,22] := 1.71608;
   DATA[161,23] := 954.8705;
   DATA[161,24] := 2.0;
   DATA[161,25] := 2.0;
   DATA[161,26] := 7.87766;
   DATA[161,27] := 145.1423;
   DATA[161,28] := 264.2271;
   DATA[161,29] := 12.26609;
   DATA[161,30] := 1.726737;
   DATA[161,31] := 1.271295;
   DATA[161,32] := 0.7348846;
   DATA[161,33] := 0.3081062;
   DATA[161,34] := 2.0;
   DATA[161,35] := 250.9933;
   DATA[161,36] := 1.585878;
   DATA[161,37] := 189.6789;
   DATA[161,38] := 0.000128152;
   DATA[161,39] := 1.0;
   DATA[162,0] := 2.555488;
   DATA[162,1] := 525.8692;
   DATA[162,2] := 2.0;
   DATA[162,3] := 2.0;
   DATA[162,4] := 262.0802;
   DATA[162,5] := 8.39163;
   DATA[162,6] := 328.2748;
   DATA[162,7] := 2.441419;
   DATA[162,8] := 2.0;
   DATA[162,9] := 2.0;
   DATA[162,10] := 2.0;
   DATA[162,11] := 19.90845;
   DATA[162,12] := 2.21324;
   DATA[162,13] := 963.4549;
   DATA[162,14] := 1.0;
   DATA[162,15] := 2.0;
   DATA[162,16] := 1.0;
   DATA[162,17] := 1.0;
   DATA[162,18] := 1.0;
   DATA[162,19] := 2.0;
   DATA[162,20] := 148.808;
   DATA[162,21] := 155.9087;
   DATA[162,22] := 1.718643;
   DATA[162,23] := 954.486;
   DATA[162,24] := 2.0;
   DATA[162,25] := 2.0;
   DATA[162,26] := 7.87766;
   DATA[162,27] := 145.1423;
   DATA[162,28] := 264.2271;
   DATA[162,29] := 12.26609;
   DATA[162,30] := 1.726737;
   DATA[162,31] := 1.290637;
   DATA[162,32] := 0.7348846;
   DATA[162,33] := 0.3066329;
   DATA[162,34] := 2.0;
   DATA[162,35] := 250.9933;
   DATA[162,36] := 1.585878;
   DATA[162,37] := 189.6789;
   DATA[162,38] := 0.000128152;
   DATA[162,39] := 1.0;
   DATA[163,0] := 2.593921;
   DATA[163,1] := 525.7907;
   DATA[163,2] := 2.0;
   DATA[163,3] := 2.0;
   DATA[163,4] := 262.0802;
   DATA[163,5] := 8.39163;
   DATA[163,6] := 328.2748;
   DATA[163,7] := 2.441419;
   DATA[163,8] := 2.0;
   DATA[163,9] := 2.0;
   DATA[163,10] := 2.0;
   DATA[163,11] := 19.90845;
   DATA[163,12] := 2.209525;
   DATA[163,13] := 963.2146;
   DATA[163,14] := 1.0;
   DATA[163,15] := 2.0;
   DATA[163,16] := 1.0;
   DATA[163,17] := 1.0;
   DATA[163,18] := 1.0;
   DATA[163,19] := 2.0;
   DATA[163,20] := 148.808;
   DATA[163,21] := 155.9087;
   DATA[163,22] := 1.718643;
   DATA[163,23] := 954.5629;
   DATA[163,24] := 2.0;
   DATA[163,25] := 2.0;
   DATA[163,26] := 7.87766;
   DATA[163,27] := 145.1423;
   DATA[163,28] := 264.2271;
   DATA[163,29] := 12.26609;
   DATA[163,30] := 1.726737;
   DATA[163,31] := 1.291789;
   DATA[163,32] := 0.7348846;
   DATA[163,33] := 0.3066329;
   DATA[163,34] := 2.0;
   DATA[163,35] := 250.9933;
   DATA[163,36] := 1.585878;
   DATA[163,37] := 189.6789;
   DATA[163,38] := 0.000128152;
   DATA[163,39] := 1.0;
   DATA[164,0] := 2.625628;
   DATA[164,1] := 525.2804;
   DATA[164,2] := 2.0;
   DATA[164,3] := 2.0;
   DATA[164,4] := 262.0802;
   DATA[164,5] := 8.39163;
   DATA[164,6] := 328.2748;
   DATA[164,7] := 2.441419;
   DATA[164,8] := 2.0;
   DATA[164,9] := 2.0;
   DATA[164,10] := 2.0;
   DATA[164,11] := 19.90845;
   DATA[164,12] := 2.209525;
   DATA[164,13] := 963.6151;
   DATA[164,14] := 1.0;
   DATA[164,15] := 2.0;
   DATA[164,16] := 1.0;
   DATA[164,17] := 1.0;
   DATA[164,18] := 1.0;
   DATA[164,19] := 2.0;
   DATA[164,20] := 148.808;
   DATA[164,21] := 155.9087;
   DATA[164,22] := 1.718643;
   DATA[164,23] := 954.14;
   DATA[164,24] := 2.0;
   DATA[164,25] := 2.0;
   DATA[164,26] := 7.87766;
   DATA[164,27] := 145.1423;
   DATA[164,28] := 264.2271;
   DATA[164,29] := 12.26609;
   DATA[164,30] := 1.726737;
   DATA[164,31] := 1.291789;
   DATA[164,32] := 0.7348846;
   DATA[164,33] := 0.3064407;
   DATA[164,34] := 2.0;
   DATA[164,35] := 250.9933;
   DATA[164,36] := 1.681991;
   DATA[164,37] := 189.6789;
   DATA[164,38] := 0.000128152;
   DATA[164,39] := 1.0;
   DATA[165,0] := 2.642923;
   DATA[165,1] := 525.0842;
   DATA[165,2] := 2.0;
   DATA[165,3] := 2.0;
   DATA[165,4] := 262.0802;
   DATA[165,5] := 8.39163;
   DATA[165,6] := 328.2748;
   DATA[165,7] := 2.441419;
   DATA[165,8] := 2.0;
   DATA[165,9] := 2.0;
   DATA[165,10] := 2.0;
   DATA[165,11] := 19.80601;
   DATA[165,12] := 2.209525;
   DATA[165,13] := 963.4149;
   DATA[165,14] := 1.0;
   DATA[165,15] := 2.0;
   DATA[165,16] := 1.0;
   DATA[165,17] := 1.0;
   DATA[165,18] := 1.0;
   DATA[165,19] := 2.0;
   DATA[165,20] := 148.808;
   DATA[165,21] := 155.9087;
   DATA[165,22] := 1.718643;
   DATA[165,23] := 953.9477;
   DATA[165,24] := 2.0;
   DATA[165,25] := 2.0;
   DATA[165,26] := 7.87766;
   DATA[165,27] := 145.1423;
   DATA[165,28] := 264.2271;
   DATA[165,29] := 12.26609;
   DATA[165,30] := 1.726737;
   DATA[165,31] := 1.291789;
   DATA[165,32] := 0.7348846;
   DATA[165,33] := 0.3068891;
   DATA[165,34] := 2.0;
   DATA[165,35] := 250.9933;
   DATA[165,36] := 1.681991;
   DATA[165,37] := 189.6789;
   DATA[165,38] := 0.000128152;
   DATA[165,39] := 1.0;
   DATA[166,0] := 2.657656;
   DATA[166,1] := 525.0056;
   DATA[166,2] := 2.0;
   DATA[166,3] := 2.0;
   DATA[166,4] := 262.0802;
   DATA[166,5] := 8.39163;
   DATA[166,6] := 328.2748;
   DATA[166,7] := 2.441547;
   DATA[166,8] := 2.0;
   DATA[166,9] := 2.0;
   DATA[166,10] := 2.0;
   DATA[166,11] := 19.7964;
   DATA[166,12] := 2.209525;
   DATA[166,13] := 963.3748;
   DATA[166,14] := 1.0;
   DATA[166,15] := 2.0;
   DATA[166,16] := 1.0;
   DATA[166,17] := 1.0;
   DATA[166,18] := 1.0;
   DATA[166,19] := 2.0;
   DATA[166,20] := 148.808;
   DATA[166,21] := 155.9087;
   DATA[166,22] := 1.718643;
   DATA[166,23] := 954.2169;
   DATA[166,24] := 2.0;
   DATA[166,25] := 2.0;
   DATA[166,26] := 7.87766;
   DATA[166,27] := 145.1423;
   DATA[166,28] := 264.2271;
   DATA[166,29] := 12.26609;
   DATA[166,30] := 1.726737;
   DATA[166,31] := 1.281798;
   DATA[166,32] := 0.7351407;
   DATA[166,33] := 0.3086186;
   DATA[166,34] := 2.0;
   DATA[166,35] := 250.9933;
   DATA[166,36] := 1.681991;
   DATA[166,37] := 189.6789;
   DATA[166,38] := 0.000128152;
   DATA[166,39] := 1.0;
   DATA[167,0] := 2.657656;
   DATA[167,1] := 524.9271;
   DATA[167,2] := 2.0;
   DATA[167,3] := 2.0;
   DATA[167,4] := 262.0802;
   DATA[167,5] := 8.39163;
   DATA[167,6] := 328.2748;
   DATA[167,7] := 2.444879;
   DATA[167,8] := 2.0;
   DATA[167,9] := 2.0;
   DATA[167,10] := 2.0;
   DATA[167,11] := 19.7964;
   DATA[167,12] := 2.209525;
   DATA[167,13] := 963.2546;
   DATA[167,14] := 1.0;
   DATA[167,15] := 2.0;
   DATA[167,16] := 1.0;
   DATA[167,17] := 1.0;
   DATA[167,18] := 1.0;
   DATA[167,19] := 2.0;
   DATA[167,20] := 148.808;
   DATA[167,21] := 155.9087;
   DATA[167,22] := 1.718643;
   DATA[167,23] := 954.2938;
   DATA[167,24] := 2.0;
   DATA[167,25] := 2.0;
   DATA[167,26] := 7.87766;
   DATA[167,27] := 145.1423;
   DATA[167,28] := 264.2271;
   DATA[167,29] := 12.26609;
   DATA[167,30] := 1.726737;
   DATA[167,31] := 1.281798;
   DATA[167,32] := 0.7360369;
   DATA[167,33] := 0.3086186;
   DATA[167,34] := 2.0;
   DATA[167,35] := 250.9933;
   DATA[167,36] := 1.681991;
   DATA[167,37] := 189.6789;
   DATA[167,38] := 0.000128152;
   DATA[167,39] := 1.0;
   DATA[168,0] := 2.634917;
   DATA[168,1] := 525.4767;
   DATA[168,2] := 2.0;
   DATA[168,3] := 2.0;
   DATA[168,4] := 262.0802;
   DATA[168,5] := 8.39163;
   DATA[168,6] := 328.2748;
   DATA[168,7] := 2.445904;
   DATA[168,8] := 2.0;
   DATA[168,9] := 2.0;
   DATA[168,10] := 2.0;
   DATA[168,11] := 19.7964;
   DATA[168,12] := 2.209525;
   DATA[168,13] := 963.3347;
   DATA[168,14] := 1.0;
   DATA[168,15] := 2.0;
   DATA[168,16] := 1.0;
   DATA[168,17] := 1.0;
   DATA[168,18] := 1.0;
   DATA[168,19] := 2.0;
   DATA[168,20] := 148.808;
   DATA[168,21] := 156.1138;
   DATA[168,22] := 1.717489;
   DATA[168,23] := 954.1784;
   DATA[168,24] := 2.0;
   DATA[168,25] := 2.0;
   DATA[168,26] := 7.875737;
   DATA[168,27] := 145.1423;
   DATA[168,28] := 264.2271;
   DATA[168,29] := 12.26609;
   DATA[168,30] := 1.726737;
   DATA[168,31] := 1.299091;
   DATA[168,32] := 0.7360369;
   DATA[168,33] := 0.3086186;
   DATA[168,34] := 2.0;
